(* IEC 61131-3 sources: verifaps-lib/share/xPPU (part 20) *)

(* ---- PLCOpenXML_Scenario_21.st ---- *)
// Extracted from file:/home/weigl/work/verifaps-lib/lang/../share/xPPU/PLCOpenXML_Scenario_21.xml on Wed Feb 05 17:44:48 CET 2020

FUNCTION_BLOCK A_to_V_Transducer

    VAR
        AI_AmperToVolt : INT;
    END_VAR

END_FUNCTION_BLOCK

FUNCTION_BLOCK BistableCylinder

    VAR_OUTPUT
        Extended : BOOL;
        Retracted : BOOL;
    END_VAR

    VAR
        DI_Extended : BOOL;
        DI_Retracted : BOOL;
        DO_Extend : BOOL;
        DO_Retract : BOOL;
        DI_BoundaryPressure : BOOL;
        DI_VacuumBoundaryPressure : BOOL;
        DI_VacuumBoundaryFlowPressure : BOOL;
        AI_PressureSensor : INT;
        AI_FlowPressure : INT;
        AI_PositionTransmitter : INT;
        SFCInit : BOOL;
        SFCReset : BOOL;
    END_VAR
    ACTION ACT_Extend

        INITIAL_STEP Init_ACT_Extend : (*Local Id: 0 *)
        END_STEP

        STEP Extend_Cylinder : (*Local Id: 3 *)
        END_STEP

        STEP SetExtended : (*Local Id: 9 *)
        END_STEP
        TRANSITION FROM (Init_ACT_Extend) TO (Extend_Cylinder) := (NOT Extended AND NOT GVL.IsSFCResetting); END_TRANSITION
        TRANSITION FROM (Extend_Cylinder) TO (SetExtended) := (DI_Extended); END_TRANSITION
        TRANSITION FROM (SetExtended) TO (Init_ACT_Extend) := (Extended); END_TRANSITION
    END_ACTION
    ACTION ACT_Retract

        INITIAL_STEP Init_ACT_Retract : (*Local Id: 0 *)
        END_STEP

        STEP Retract_Cylinder : (*Local Id: 3 *)
        END_STEP

        STEP SetRetacted : (*Local Id: 9 *)
        END_STEP
        TRANSITION FROM (Init_ACT_Retract) TO (Retract_Cylinder) := (NOT Retracted AND NOT GVL.IsSFCResetting); END_TRANSITION
        TRANSITION FROM (Retract_Cylinder) TO (SetRetacted) := (DI_Retracted); END_TRANSITION
        TRANSITION FROM (SetRetacted) TO (Init_ACT_Retract) := (Retracted); END_TRANSITION
    END_ACTION

END_FUNCTION_BLOCK

FUNCTION_BLOCK Crane

    VAR_INPUT
        LiftingCylinder : MonostableCylinder;
        Gripper : VacuumGripper;
        Table : TurningTable;
        SoftwareEmergency : BOOL;
        Check_Stack_WPProvided : BOOL;
        Check_Stack_WPType_Black : BOOL;
        Check_Stack_WPType_White : BOOL;
        Check_Stack_WPType_Metallic : BOOL;
        Check_LargeSortingConveyor_IsSorting : BOOL;
        Check_LargeSortingConveyor_AutomaticExecuteCompleted : BOOL;
        Check_Stamp_IsStamping : BOOL;
        Check_Stamp_WPAvailable : BOOL;
        Check_Stamp_AutomaticExecuteCompleted : BOOL;
        Check_RefillConveyor_IsSending : BOOL;
        Check_EngineStop : BOOL;
        SFCReset : BOOL;
    END_VAR

    VAR_OUTPUT
        InitCompleted : BOOL;
        AutomaticExecuteCompleted : BOOL;
        Conveyor_AllowedToOperate : BOOL;
        Stamp_AllowedToOperate : BOOL;
        WPPickedUp : BOOL;
        EmergencyHandled : BOOL;
    END_VAR

    VAR
        CraneSpeed : INT;
        WPPutDown : BOOL;
        ReachedStack : BOOL;
        ReachedConveyor : BOOL;
        ReachedStamp : BOOL;
        WPType_White : BOOL;
        WPType_Black : BOOL;
        WPType_Metallic : BOOL;
        WPWeight_Light : BOOL;
        WPWeight_Medium : BOOL;
        WPWeight_Heavy : BOOL;
        SFCInit : BOOL;
    END_VAR
    ACTION Reset_ConveyorAllowedToOperate

        Conveyor_AllowedToOperate := FALSE;
    END_ACTION
    ACTION Reset_StampAllowedToOperate

        Stamp_AllowedToOperate := FALSE;
    END_ACTION
    ACTION Reset_Variables

        InitCompleted := FALSE;
        AutomaticExecuteCompleted := FALSE;
        Conveyor_AllowedToOperate := FALSE;
        Stamp_AllowedToOperate := FALSE;

        WPPickedUp := FALSE;
        WPPutDown := FALSE;
        ReachedStack := FALSE;
        ReachedConveyor := FALSE;
        ReachedStamp := FALSE;
        WPType_White := FALSE;
        WPType_Black := FALSE;
        WPType_Metallic := FALSE;
        WPWeight_Light := FALSE;
        WPWeight_Medium := FALSE;
        WPWeight_Heavy := FALSE;
    END_ACTION
    ACTION Set_ConveyorAllowedToOperate

        Conveyor_AllowedToOperate := TRUE;
    END_ACTION
    ACTION Set_StampAllowedToOperate

        Stamp_AllowedToOperate := TRUE;
    END_ACTION
    ACTION Set_WPTypeEqualsStack

        WPType_White:=Main.Stack_WPType_White;
        WPType_Black:=Main.Stack_WPType_Black;
        WPType_Metallic:=Main.Stack_WPType_Metallic;
        WPWeight_Light:=Main.Stack_WPWeight_Light;
        WPWeight_Medium:=Main.Stack_WPWeight_Medium;
        WPWeight_Heavy:=Main.Stack_WPWeight_Heavy;
    END_ACTION
    ACTION Set_WPTypeEqualsStamp

        WPType_White:=Main.Stamp_WPType_White;
        WPType_Black:=Main.Stamp_WPType_Black;
        WPType_Metallic:=Main.Stamp_WPType_Metallic;
        WPWeight_Light:=Main.Stamp_WPWeight_Light;
        WPWeight_Medium:=Main.Stamp_WPWeight_Medium;
        WPWeight_Heavy:=Main.Stamp_WPWeight_Heavy;
    END_ACTION
    ACTION ACT_MoveToConveyor

        INITIAL_STEP Init_MoveToConveyor : (*Local Id: 0 *)
        END_STEP

        STEP DecideHowToMoveCrane : (*Local Id: 3 *)
        END_STEP

        STEP Turn_CounterClockwise_MTC : (*Local Id: 7 *)
            Table.Motor.ACT_TurnCounterclockwise(N);
        END_STEP

        STEP Turn_CLockwise_MTC : (*Local Id: 13 *)
            Table.Motor.ACT_TurnClockwise(N);
        END_STEP

        STEP First_Turn_CounterC : (*Local Id: 18 *)
            Table.Motor.ACT_TurnCounterclockwise(N);
        END_STEP

        STEP Second_Turn_Clockwise : (*Local Id: 24 *)
            Table.Motor.ACT_TurnClockwise(N);
        END_STEP

        STEP StopCrane : (*Local Id: 30 *)
            Table.Motor.ACT_Stop(N);
        END_STEP

        STEP SetReachedConveyor : (*Local Id: 33 *)
        END_STEP
        TRANSITION FROM (DecideHowToMoveCrane) TO (Turn_CounterClockwise_MTC) := (Table.AtStack.DI_SwitchTrue); END_TRANSITION
        TRANSITION FROM (DecideHowToMoveCrane) TO (Turn_CLockwise_MTC) := (Table.AtStamp.DI_SwitchTrue); END_TRANSITION
        TRANSITION FROM (DecideHowToMoveCrane) TO (First_Turn_CounterC) := (NOT (Table.AtStack.DI_SwitchTrue AND Table.AtStamp.DI_SwitchTrue)); END_TRANSITION
        TRANSITION FROM (DecideHowToMoveCrane) TO (Turn_CLockwise_MTC) := (Table.AtStamp.DI_SwitchTrue); END_TRANSITION
        TRANSITION FROM (DecideHowToMoveCrane) TO (First_Turn_CounterC) := (NOT (Table.AtStack.DI_SwitchTrue AND Table.AtStamp.DI_SwitchTrue)); END_TRANSITION
        TRANSITION FROM (First_Turn_CounterC) TO (StopCrane) := (Table.AtConveyor.DI_SwitchTrue); END_TRANSITION
        TRANSITION FROM (First_Turn_CounterC) TO (Second_Turn_Clockwise) := (First_Turn_CounterC.t>T#8s AND Not Table.AtConveyor.DI_SwitchTrue); END_TRANSITION
        TRANSITION FROM (First_Turn_CounterC) TO (StopCrane) := (Table.AtConveyor.DI_SwitchTrue); END_TRANSITION
        TRANSITION FROM (Second_Turn_Clockwise) TO (StopCrane) := (Table.AtConveyor.DI_SwitchTrue); END_TRANSITION
        TRANSITION FROM (Turn_CLockwise_MTC) TO (StopCrane) := (Table.AtConveyor.DI_SwitchTrue); END_TRANSITION
        TRANSITION FROM (First_Turn_CounterC) TO (StopCrane) := (Table.AtConveyor.DI_SwitchTrue); END_TRANSITION
        TRANSITION FROM (Second_Turn_Clockwise) TO (StopCrane) := (Table.AtConveyor.DI_SwitchTrue); END_TRANSITION
        TRANSITION FROM (Turn_CounterClockwise_MTC) TO (StopCrane) := (Table.AtConveyor.DI_SwitchTrue); END_TRANSITION
        TRANSITION FROM (Turn_CLockwise_MTC) TO (StopCrane) := (Table.AtConveyor.DI_SwitchTrue); END_TRANSITION
        TRANSITION FROM (First_Turn_CounterC) TO (StopCrane) := (Table.AtConveyor.DI_SwitchTrue); END_TRANSITION
        TRANSITION FROM (Second_Turn_Clockwise) TO (StopCrane) := (Table.AtConveyor.DI_SwitchTrue); END_TRANSITION
        TRANSITION FROM (Init_MoveToConveyor) TO (DecideHowToMoveCrane) := (NOT GVL.IsSFCResetting); END_TRANSITION
        TRANSITION FROM (StopCrane) TO (SetReachedConveyor) := (Table.Motor.Stopped); END_TRANSITION
        TRANSITION FROM (SetReachedConveyor) TO (Init_MoveToConveyor) := (ReachedConveyor); END_TRANSITION
    END_ACTION
    ACTION ACT_MoveToStack

        INITIAL_STEP Init_MoveToMagazine : (*Local Id: 0 *)
        END_STEP

        STEP Turn_Clockwise_MTM : (*Local Id: 3 *)
            Table.Motor.ACT_TurnClockwise(N);
        END_STEP

        STEP Turn_Counterclockwise : (*Local Id: 9 *)
            Table.Motor.ACT_TurnCounterclockwise(N);
        END_STEP

        STEP StopCrane : (*Local Id: 13 *)
            Table.Motor.ACT_Stop(N);
        END_STEP

        STEP SetReachedStack : (*Local Id: 16 *)
        END_STEP
        TRANSITION FROM (Turn_Clockwise_MTM) TO (StopCrane) := (Table.AtStack.DI_SwitchTrue); END_TRANSITION
        TRANSITION FROM (Turn_Clockwise_MTM) TO (Turn_Counterclockwise) := (Turn_Clockwise_MTM.t>T#8s); END_TRANSITION
        TRANSITION FROM (Turn_Clockwise_MTM) TO (StopCrane) := (Table.AtStack.DI_SwitchTrue); END_TRANSITION
        TRANSITION FROM (Turn_Counterclockwise) TO (StopCrane) := (Table.AtStack.DI_SwitchTrue); END_TRANSITION
        TRANSITION FROM (Init_MoveToMagazine) TO (Turn_Clockwise_MTM) := (NOT GVL.IsSFCResetting); END_TRANSITION
        TRANSITION FROM (StopCrane) TO (SetReachedStack) := (Table.Motor.Stopped); END_TRANSITION
        TRANSITION FROM (SetReachedStack) TO (Init_MoveToMagazine) := (ReachedStack); END_TRANSITION
    END_ACTION
    ACTION ACT_MoveToStamp

        INITIAL_STEP Init_MoveToStamp : (*Local Id: 0 *)
        END_STEP

        STEP Turn_CounterClockwise_MTS : (*Local Id: 3 *)
            Table.Motor.ACT_TurnCounterclockwise(N);
        END_STEP

        STEP Turn_Clockwise : (*Local Id: 9 *)
            Table.Motor.ACT_TurnClockwise(N);
        END_STEP

        STEP StopCrane : (*Local Id: 13 *)
            Table.Motor.ACT_Stop(N);
        END_STEP

        STEP SetReachedStamp : (*Local Id: 16 *)
        END_STEP
        TRANSITION FROM (Turn_CounterClockwise_MTS) TO (StopCrane) := (Table.AtStamp.DI_SwitchTrue); END_TRANSITION
        TRANSITION FROM (Turn_CounterClockwise_MTS) TO (Turn_Clockwise) := (Turn_CounterClockwise_MTS.t>T#8s); END_TRANSITION
        TRANSITION FROM (Turn_CounterClockwise_MTS) TO (StopCrane) := (Table.AtStamp.DI_SwitchTrue); END_TRANSITION
        TRANSITION FROM (Turn_Clockwise) TO (StopCrane) := (Table.AtStamp.DI_SwitchTrue); END_TRANSITION
        TRANSITION FROM (Init_MoveToStamp) TO (Turn_CounterClockwise_MTS) := (NOT GVL.IsSFCResetting); END_TRANSITION
        TRANSITION FROM (StopCrane) TO (SetReachedStamp) := (Table.Motor.Stopped); END_TRANSITION
        TRANSITION FROM (SetReachedStamp) TO (Init_MoveToStamp) := (ReachedStamp); END_TRANSITION
    END_ACTION
    ACTION ACT_PickUpWP

        INITIAL_STEP Init_PickUpWP : (*Local Id: 0 *)
        END_STEP

        STEP Crane_Down : (*Local Id: 3 *)
            LiftingCylinder.ACT_Extend(N);
        END_STEP

        STEP SetWPType : (*Local Id: 6 *)
        END_STEP

        STEP WPType_Is_WPTypeStack : (*Local Id: 10 *)
            Set_WPTypeEqualsStack(N);
        END_STEP

        STEP WPType_Is_WPTypeStamp : (*Local Id: 15 *)
            Set_WPTypeEqualsStamp(N);
        END_STEP

        STEP Turn_On_Vacuum_PWU : (*Local Id: 19 *)
            Gripper.ACT_Intake(N);
        END_STEP

        STEP Crane_Up : (*Local Id: 23 *)
            LiftingCylinder.ACT_Retract(N);
        END_STEP

        STEP Error : (*Local Id: 28 *)
        END_STEP

        STEP SetWPPickedUp : (*Local Id: 35 *)
        END_STEP
        TRANSITION FROM (SetWPType) TO (WPType_Is_WPTypeStack) := (ReachedStack); END_TRANSITION
        TRANSITION FROM (SetWPType) TO (WPType_Is_WPTypeStamp) := (ReachedStamp); END_TRANSITION
        TRANSITION FROM (Turn_On_Vacuum_PWU) TO (Crane_Up) := (Gripper.Intaken); END_TRANSITION
        TRANSITION FROM (Turn_On_Vacuum_PWU) TO (Error) := (Turn_On_Vacuum_PWU.t>T#2s AND NOT Gripper.Intaken); END_TRANSITION
        TRANSITION FROM (WPType_Is_WPTypeStack) TO (Turn_On_Vacuum_PWU) := (WPWeight_Heavy=Main.Stack_WPWeight_Heavy); END_TRANSITION
        TRANSITION FROM (WPType_Is_WPTypeStamp) TO (Turn_On_Vacuum_PWU) := (WPWeight_Heavy=Main.Stamp_WPWeight_Heavy); END_TRANSITION
        TRANSITION FROM (Crane_Up) TO (SetWPPickedUp) := (LiftingCylinder.Retracted); END_TRANSITION
        TRANSITION FROM (Init_PickUpWP) TO (Crane_Down) := (NOT GVL.IsSFCResetting); END_TRANSITION
        TRANSITION FROM (Crane_Down) TO (SetWPType) := (LiftingCylinder.Extended); END_TRANSITION
        TRANSITION FROM (Error) TO (Init_PickUpWP) := (SoftwareEmergency); END_TRANSITION
        TRANSITION FROM (SetWPPickedUp) TO (Init_PickUpWP) := (WPPickedUp); END_TRANSITION
    END_ACTION
    ACTION ACT_PutDownWP

        INITIAL_STEP Init_PutWPDown : (*Local Id: 0 *)
        END_STEP

        STEP WPWeight_Choice : (*Local Id: 3 *)
        END_STEP

        STEP WPLight : (*Local Id: 7 *)
        END_STEP

        STEP WPMedium : (*Local Id: 12 *)
        END_STEP

        STEP WPHeavy : (*Local Id: 17 *)
        END_STEP

        STEP Lower_Crane_PWD : (*Local Id: 21 *)
            LiftingCylinder.ACT_Extend(N);
        END_STEP

        STEP Put_WP_Down_1 : (*Local Id: 24 *)
            Gripper.ACT_Release(N);
        END_STEP

        STEP Crane_Up : (*Local Id: 27 *)
            LiftingCylinder.ACT_Retract(N);
        END_STEP

        STEP SetWPPutDown : (*Local Id: 30 *)
        END_STEP
        TRANSITION FROM (WPWeight_Choice) TO (WPLight) := (WPWeight_Light); END_TRANSITION
        TRANSITION FROM (WPWeight_Choice) TO (WPMedium) := (WPWeight_Medium); END_TRANSITION
        TRANSITION FROM (WPWeight_Choice) TO (WPHeavy) := (WPWeight_Heavy); END_TRANSITION
        TRANSITION FROM (WPLight) TO (Lower_Crane_PWD) := (WPLight.t>T#0ms); END_TRANSITION
        TRANSITION FROM (WPMedium) TO (Lower_Crane_PWD) := (WPMedium.t>T#1000ms); END_TRANSITION
        TRANSITION FROM (WPHeavy) TO (Lower_Crane_PWD) := (WPHeavy.t>T#2000ms); END_TRANSITION
        TRANSITION FROM (Init_PutWPDown) TO (WPWeight_Choice) := (NOT GVL.IsSFCResetting); END_TRANSITION
        TRANSITION FROM (Lower_Crane_PWD) TO (Put_WP_Down_1) := (LiftingCylinder.Extended); END_TRANSITION
        TRANSITION FROM (Put_WP_Down_1) TO (Crane_Up) := (Gripper.Released); END_TRANSITION
        TRANSITION FROM (Crane_Up) TO (SetWPPutDown) := (LiftingCylinder.Retracted); END_TRANSITION
        TRANSITION FROM (SetWPPutDown) TO (Init_PutWPDown) := (WPPutDown); END_TRANSITION
    END_ACTION
    ACTION ACT_AutomaticExecute

        INITIAL_STEP ACT_AutomaticExecute_Init : (*Local Id: 0 *)
        END_STEP

        STEP Waiting_For_Stack_To_Provide_WP : (*Local Id: 3 *)
        END_STEP

        STEP Check_WP_Type : (*Local Id: 6 *)
        END_STEP

        STEP Crane_To_Stamp_1 : (*Local Id: 10 *)
            ACT_MoveToStack(N);
        END_STEP

        STEP Pick_Up_WP_1 : (*Local Id: 13 *)
            ACT_PickUpWP(N);
        END_STEP

        STEP Check_RC_1 : (*Local Id: 16 *)
        END_STEP

        STEP Crane_Turning_To_Conveyor_1 : (*Local Id: 19 *)
            ACT_MoveToConveyor(N);
        END_STEP

        STEP Putting_Down_WP_1 : (*Local Id: 22 *)
            ACT_PutDownWP(N);
        END_STEP

        STEP Short_Delay : (*Local Id: 25 *)
        END_STEP

        STEP Sort_WP : (*Local Id: 28 *)
            Set_ConveyorAllowedToOperate(P0);
            Reset_ConveyorAllowedToOperate(P1);
        END_STEP

        STEP CheckStamp_WPAvailable : (*Local Id: 31 *)
        END_STEP

        STEP WP_Should_Be_Stamped : (*Local Id: 41 *)
        END_STEP

        STEP Crane_Turning_To_Stack_1 : (*Local Id: 45 *)
            ACT_MoveToStack(N);
        END_STEP

        STEP Crane_Pick_Up_Wp_2 : (*Local Id: 48 *)
            ACT_PickUpWP(N);
        END_STEP

        STEP Check_RC_2 : (*Local Id: 51 *)
        END_STEP

        STEP Crane_Turning_To_Stamp_2 : (*Local Id: 54 *)
            ACT_MoveToStamp(N);
        END_STEP

        STEP Crane_Put_Down_WP_2 : (*Local Id: 57 *)
            ACT_PutDownWP(N);
        END_STEP

        STEP Stamping_WP : (*Local Id: 60 *)
            Set_StampAllowedToOperate(P0);
        END_STEP

        STEP CheckStamp_AutomaticExecuteCompleted : (*Local Id: 68 *)
            Reset_StampAllowedToOperate(P1);
        END_STEP

        STEP Crane_Turning_To_Stamp_3 : (*Local Id: 73 *)
            ACT_MoveToStamp(N);
        END_STEP
        TRANSITION FROM (Check_WP_Type) TO (Crane_To_Stamp_1) := (Check_Stack_WPType_Black); END_TRANSITION
        TRANSITION FROM (Check_WP_Type) TO (WP_Should_Be_Stamped) := (Check_Stack_WPType_Metallic OR Check_Stack_WPType_White); END_TRANSITION
        TRANSITION FROM (CheckStamp_WPAvailable) TO (Waiting_For_Stack_To_Provide_WP) := (NOT Check_Stamp_WPAvailable); END_TRANSITION
        TRANSITION FROM (CheckStamp_WPAvailable) TO (Crane_Turning_To_Stamp_3) := (Check_Stamp_WPAvailable); END_TRANSITION
        TRANSITION FROM (WP_Should_Be_Stamped) TO (Crane_Turning_To_Stack_1) := (NOT Check_Stamp_IsStamping); END_TRANSITION
        TRANSITION FROM (WP_Should_Be_Stamped) TO (Crane_Turning_To_Stamp_3) := (Check_Stamp_IsStamping); END_TRANSITION
        TRANSITION FROM (Stamping_WP) TO (CheckStamp_AutomaticExecuteCompleted) := (Check_Stack_WPType_Metallic OR Check_Stack_WPType_White); END_TRANSITION
        TRANSITION FROM (Stamping_WP) TO (Crane_To_Stamp_1) := (Check_Stack_WPType_Black); END_TRANSITION
        TRANSITION FROM (CheckStamp_WPAvailable) TO (Waiting_For_Stack_To_Provide_WP) := (NOT Check_Stamp_WPAvailable); END_TRANSITION
        TRANSITION FROM (Stamping_WP) TO (CheckStamp_AutomaticExecuteCompleted) := (Check_Stack_WPType_Metallic OR Check_Stack_WPType_White); END_TRANSITION
        TRANSITION FROM (CheckStamp_AutomaticExecuteCompleted) TO (Pick_Up_WP_1) := (Check_Stamp_AutomaticExecuteCompleted); END_TRANSITION
        TRANSITION FROM (Crane_Turning_To_Stamp_3) TO (Pick_Up_WP_1) := (ReachedStamp AND NOT Check_Stamp_AutomaticExecuteCompleted); END_TRANSITION
        TRANSITION FROM (CheckStamp_WPAvailable) TO (Waiting_For_Stack_To_Provide_WP) := (NOT Check_Stamp_WPAvailable); END_TRANSITION
        TRANSITION FROM (ACT_AutomaticExecute_Init) TO (Waiting_For_Stack_To_Provide_WP) := (NOT AutomaticExecuteCompleted AND NOT GVL.IsSFCResetting); END_TRANSITION
        TRANSITION FROM (Waiting_For_Stack_To_Provide_WP) TO (Check_WP_Type) := (Check_Stack_WPProvided); END_TRANSITION
        TRANSITION FROM (Crane_To_Stamp_1) TO (Pick_Up_WP_1) := (ReachedStack); END_TRANSITION
        TRANSITION FROM (Pick_Up_WP_1) TO (Check_RC_1) := (WPPickedUp); END_TRANSITION
        TRANSITION FROM (Check_RC_1) TO (Crane_Turning_To_Conveyor_1) := (NOT Check_RefillConveyor_IsSending AND Check_Rc_1.t>T#250ms); END_TRANSITION
        TRANSITION FROM (Crane_Turning_To_Conveyor_1) TO (Putting_Down_WP_1) := (ReachedConveyor AND NOT Check_LargeSortingConveyor_IsSorting); END_TRANSITION
        TRANSITION FROM (Putting_Down_WP_1) TO (Short_Delay) := (WPPutDown); END_TRANSITION
        TRANSITION FROM (Short_Delay) TO (Sort_WP) := (Short_Delay.t>T#50ms); END_TRANSITION
        TRANSITION FROM (Sort_WP) TO (CheckStamp_WPAvailable) := (Check_LargeSortingConveyor_AutomaticExecuteCompleted); END_TRANSITION
        TRANSITION FROM (Crane_Turning_To_Stack_1) TO (Crane_Pick_Up_Wp_2) := (ReachedStack); END_TRANSITION
        TRANSITION FROM (Crane_Pick_Up_Wp_2) TO (Check_RC_2) := (WPPickedUp); END_TRANSITION
        TRANSITION FROM (Check_RC_2) TO (Crane_Turning_To_Stamp_2) := (NOT Check_RefillConveyor_IsSending AND Check_Rc_2.t>T#250ms); END_TRANSITION
        TRANSITION FROM (Crane_Turning_To_Stamp_2) TO (Crane_Put_Down_WP_2) := (ReachedStamp); END_TRANSITION
        TRANSITION FROM (Crane_Put_Down_WP_2) TO (Stamping_WP) := (WPPutDown); END_TRANSITION
    END_ACTION
    ACTION ACT_EmergencyStop

        INITIAL_STEP Crane_ACT_EmergencyStop_Init : (*Local Id: 0 *)
        END_STEP

        STEP ResetVariables : (*Local Id: 3 *)
            Reset_Variables(N);
        END_STEP

        STEP StopCrane : (*Local Id: 6 *)
            Table.Motor.ACT_Stop(N);
        END_STEP

        STEP Turn_Vacuum_Off : (*Local Id: 12 *)
            Gripper.ACT_Release(N);
        END_STEP

        STEP Retract_LiftingCylinder : (*Local Id: 16 *)
            LiftingCylinder.ACT_Retract(N);
        END_STEP

        STEP Crane_EmergencyHandled : (*Local Id: 19 *)
        END_STEP
        TRANSITION FROM (StopCrane) TO (Retract_LiftingCylinder) := (Table.Motor.Stopped AND Gripper.Intaken); END_TRANSITION
        TRANSITION FROM (StopCrane) TO (Turn_Vacuum_Off) := (Table.Motor.Stopped AND NOT Gripper.Intaken); END_TRANSITION
        TRANSITION FROM (StopCrane) TO (Retract_LiftingCylinder) := (Table.Motor.Stopped AND Gripper.Intaken); END_TRANSITION
        TRANSITION FROM (Turn_Vacuum_Off) TO (Retract_LiftingCylinder) := (Gripper.Released); END_TRANSITION
        TRANSITION FROM (Crane_ACT_EmergencyStop_Init) TO (ResetVariables) := (NOT EmergencyHandled AND NOT GVL.IsSFCResetting); END_TRANSITION
        TRANSITION FROM (ResetVariables) TO (StopCrane) := (NOT InitCompleted AND NOT AutomaticExecuteCompleted); END_TRANSITION
        TRANSITION FROM (Retract_LiftingCylinder) TO (Crane_EmergencyHandled) := (LiftingCylinder.Retracted); END_TRANSITION
        TRANSITION FROM (Crane_EmergencyHandled) TO (Crane_ACT_EmergencyStop_Init) := (EmergencyHandled); END_TRANSITION
    END_ACTION
    ACTION ACT_Init

        INITIAL_STEP Crane_ACT_Init : (*Local Id: 0 *)
        END_STEP

        STEP Crane_MoveUp_Init : (*Local Id: 3 *)
            LiftingCylinder.ACT_Retract(N);
        END_STEP

        STEP WPAllreadyPickedUp : (*Local Id: 9 *)
        END_STEP

        STEP Turn_To_Conveyor : (*Local Id: 14 *)
            ACT_MoveToConveyor(N);
        END_STEP

        STEP Put_WP_On_Conveyor_Init : (*Local Id: 17 *)
            ACT_PutDownWP(N);
        END_STEP

        STEP Is_WP_At_Stamp : (*Local Id: 23 *)
        END_STEP

        STEP Turn_To_Stamp_Init : (*Local Id: 29 *)
            ACT_MoveToStamp(N);
        END_STEP

        STEP PicWPFromStampUp : (*Local Id: 32 *)
            ACT_PickUpWP(N);
        END_STEP

        STEP SetInitCompleted : (*Local Id: 37 *)
        END_STEP
        TRANSITION FROM (Crane_MoveUp_Init) TO (Is_WP_At_Stamp) := (LiftingCylinder.Retracted AND NOT Gripper.VacuumSwitch.DI_TakenIn); END_TRANSITION
        TRANSITION FROM (Crane_MoveUp_Init) TO (WPAllreadyPickedUp) := (LiftingCylinder.Retracted AND Gripper.VacuumSwitch.DI_TakenIn); END_TRANSITION
        TRANSITION FROM (Is_WP_At_Stamp) TO (SetInitCompleted) := (NOT Check_Stamp_WPAvailable); END_TRANSITION
        TRANSITION FROM (Is_WP_At_Stamp) TO (Turn_To_Stamp_Init) := (Check_Stamp_WPAvailable); END_TRANSITION
        TRANSITION FROM (Crane_MoveUp_Init) TO (Is_WP_At_Stamp) := (LiftingCylinder.Retracted AND NOT Gripper.VacuumSwitch.DI_TakenIn); END_TRANSITION
        TRANSITION FROM (Put_WP_On_Conveyor_Init) TO (Is_WP_At_Stamp) := (WPPutDown); END_TRANSITION
        TRANSITION FROM (Is_WP_At_Stamp) TO (SetInitCompleted) := (NOT Check_Stamp_WPAvailable); END_TRANSITION
        TRANSITION FROM (Crane_ACT_Init) TO (Crane_MoveUp_Init) := (NOT InitCompleted AND NOT GVL.IsSFCResetting); END_TRANSITION
        TRANSITION FROM (WPAllreadyPickedUp) TO (Turn_To_Conveyor) := (WPPickedUp); END_TRANSITION
        TRANSITION FROM (Turn_To_Conveyor) TO (Put_WP_On_Conveyor_Init) := (ReachedConveyor); END_TRANSITION
        TRANSITION FROM (Turn_To_Stamp_Init) TO (PicWPFromStampUp) := (ReachedStamp); END_TRANSITION
        TRANSITION FROM (PicWPFromStampUp) TO (Turn_To_Conveyor) := (WPPickedUp); END_TRANSITION
        TRANSITION FROM (SetInitCompleted) TO (Crane_ACT_Init) := (InitCompleted); END_TRANSITION
    END_ACTION

    Check_Stack_WPProvided := Main.Stack_WPProvided;
    Check_Stack_WPType_Black := Main.Stack_WPType_Black;
    Check_Stack_WPType_White := Main.Stack_WPType_White;
    Check_Stack_WPType_Metallic := Main.Stack_WPType_Metallic;
    Check_LargeSortingConveyor_IsSorting := Main.LargeSortingConveyor_IsSorting;
    Check_LargeSortingConveyor_AutomaticExecuteCompleted := Main.LargeSortingConveyor_AutomaticExecuteCompleted;
    Check_Stamp_IsStamping := Main.Stamp_IsStamping;
    Check_Stamp_WPAvailable := Main.Stamp_WPAvailable;
    Check_Stamp_AutomaticExecuteCompleted := Main.Stamp_AutomaticExecuteCompleted;
    Check_RefillConveyor_IsSending := Main.Check_RefillConveyor_IsSending;
    Check_EngineStop := MAIN.PPU_EngineStop;
    IF Check_EngineStop THEN
    	Table.Motor.ACT_Stop();
    END_IF
END_FUNCTION_BLOCK

FUNCTION_BLOCK EnergyMonitor

    VAR
        BK_1_6_Wattmeter : Wattmeter;
        BK_2_3_7_Wattmeter : Wattmeter;
        BK_4_5_8_9_10_11_Wattmeter : Wattmeter;
        GearPoint_80l_min : GearPointFlowSensor;
        GearPoint_120l_min : GearPointFlowSensor;
        PressureSensor_4bar : PressureSensor_4bar;
        Flow_2to200l_min : FlowSensor;
        Transducer_0to10AC_0to10V : A_to_V_Transducer;
        ExtSensor_0to10V : V_Sensor;
        PressureSensor : PressureSensor;
        SmallContacter_left : ProtectiveContact;
        SmallContacter_right : ProtectiveContact;
        ChangeoverMagnetVaveRelay : MagnetValve;
    END_VAR

END_FUNCTION_BLOCK

FUNCTION_BLOCK FlowSensor

    VAR
        AI_Flow : INT;
    END_VAR

END_FUNCTION_BLOCK

FUNCTION_BLOCK GearPointFlowSensor

    VAR
        DI_ReachedGearPoint : BOOL;
    END_VAR

END_FUNCTION_BLOCK

FUNCTION_BLOCK InductiveSensor

    VAR
        DI_WPMetallic : BOOL;
    END_VAR

END_FUNCTION_BLOCK

FUNCTION_BLOCK InductiveSwitch

    VAR
        DI_InductiveSwitchTrue : BOOL;
    END_VAR

END_FUNCTION_BLOCK

FUNCTION_BLOCK LargeSortingConveyor

    VAR_INPUT
        Panel : OperationPanel;
        Motor : Motor;
        Seperator1 : MonostableCylinder;
        Seperator2 : MonostableCylinder;
        PsBeginning : PresenceSensor;
        OptRamp1 : OpticalSensor;
        IndRamp1 : InductiveSensor;
        Ramp1 : Ramp;
        UltrasonicSensor : UltrasonicSensor;
        Switch : Switch;
        OptRamp2 : OpticalSensor;
        IndRamp2 : InductiveSensor;
        Ramp2 : Ramp;
        OptEnd : OpticalSensor;
        Ramp3 : Ramp;
        OptBeginning : OpticalSensor;
        Check_AllowedToOperate : BOOL;
        Check_FollowConveyorInitCompleted : BOOL;
        Check_FollowConveyorAutoamticExecuteCompleted : BOOL;
        Check_EngineStop : BOOL;
        SFCReset : BOOL;
    END_VAR

    VAR_OUTPUT
        StartButton : BOOL;
        ManuelMode : BOOL;
        AutomaticMode : BOOL;
        InitCompleted : BOOL;
        FollowConveyor_AllowedToInit : BOOL;
        FollowConveyor_AllowedToOperate : BOOL;
        NumberOfWPsAtConveyor : USINT;
        AutomaticExecuteCompleted : BOOL;
        EmergencyStop : BOOL;
        EmergencyHandled : BOOL;
        IsSorting : BOOL;
    END_VAR

    VAR
        ConveyorSpeed : INT;
        WPSorted : BOOL;
        WPTypeChecked : BOOL;
        TargetChanged : BOOL;
        WPType_White : BOOL;
        WPType_Black : BOOL;
        WPType_Metallic : BOOL;
        CurrentTarget_Ramp1 : BOOL;
        CurrentTarget_Conveyor : BOOL;
        CurrentTarget_Ramp2 : BOOL;
        CurrentTarget_Ramp3 : BOOL;
        Priority_White : UINT;
        Priority_Black : UINT;
        Priority_Metallic : UINT;
        SFCInit : BOOL;
    END_VAR
    ACTION Reset_FollowConveyorAllowedToOperate

        FollowConveyor_AllowedToOperate := FALSE;
    END_ACTION
    ACTION Reset_Variables

        InitCompleted := FALSE;
        FollowConveyor_AllowedToInit := FALSE;
        FollowConveyor_AllowedToOperate := FALSE;
        AutomaticExecuteCompleted := FALSE;
        IsSorting:=FALSE;

        WPSorted:=FALSE;
        WPTypeChecked:=FALSE;
        TargetChanged:=FALSE;
        WPType_White:=FALSE;
        WPType_Black:=FALSE;
        WPType_Metallic:=FALSE;
        CurrentTarget_Ramp1:=FALSE;
        CurrentTarget_Conveyor:=FALSE;
        CurrentTarget_Ramp2:=FALSE;
        CurrentTarget_Ramp3:=FALSE;
    END_ACTION
    ACTION Set_FollowConveyorAllowedToOperate

        FollowConveyor_AllowedToOperate := TRUE;
    END_ACTION
    ACTION Set_OneWP

        NumberOfWPsAtConveyor:=1;
    END_ACTION
    ACTION Set_PriorityBlack

        Priority_Black := 4;
    END_ACTION
    ACTION Set_PriorityMetallic

        Priority_Metallic := 3;
    END_ACTION
    ACTION Set_PriorityWhite

        Priority_White := 1;
    END_ACTION
    ACTION Set_ThreeWP

        NumberOfWPsAtConveyor:=3;
    END_ACTION
    ACTION Set_TwoWP

        NumberOfWPsAtConveyor:=2;
    END_ACTION
    ACTION Set_ZeroWP

        NumberOfWPsAtConveyor:=0;
    END_ACTION
    ACTION ACT_ChangeTarget

        INITIAL_STEP ACT_ChangeTarget_Init : (*Local Id: 0 *)
        END_STEP

        STEP ResetTargets : (*Local Id: 3 *)
        END_STEP

        STEP White : (*Local Id: 13 *)
            Set_PriorityWhite(N);
        END_STEP

        STEP Ramp_1 : (*Local Id: 17 *)
        END_STEP

        STEP Choice_Ramp1Full : (*Local Id: 35 *)
        END_STEP

        STEP Conveyor : (*Local Id: 41 *)
        END_STEP

        STEP Black : (*Local Id: 52 *)
            Set_PriorityBlack(N);
        END_STEP

        STEP Ramp_2 : (*Local Id: 56 *)
        END_STEP

        STEP Choice_Ramp2Full : (*Local Id: 74 *)
        END_STEP

        STEP Metallic : (*Local Id: 86 *)
            Set_PriorityMetallic(N);
        END_STEP

        STEP Ramp_3 : (*Local Id: 90 *)
        END_STEP

        STEP Choice_Ramp3Full : (*Local Id: 105 *)
        END_STEP

        STEP SetTargetChanged : (*Local Id: 115 *)
        END_STEP
        TRANSITION FROM (ResetTargets) TO (White) := (WPType_White); END_TRANSITION
        TRANSITION FROM (ResetTargets) TO (Black) := (WPType_Black); END_TRANSITION
        TRANSITION FROM (ResetTargets) TO (Metallic) := (WPType_Metallic); END_TRANSITION
        TRANSITION FROM (ResetTargets) TO (White) := (WPType_White); END_TRANSITION
        TRANSITION FROM (ResetTargets) TO (Black) := (WPType_Black); END_TRANSITION
        TRANSITION FROM (White) TO (Ramp_1) := (Priority_White=1); END_TRANSITION
        TRANSITION FROM (White) TO (Ramp_2) := (Priority_White=2); END_TRANSITION
        TRANSITION FROM (White) TO (Ramp_3) := (Priority_White=3); END_TRANSITION
        TRANSITION FROM (White) TO (Conveyor) := (Priority_White=4); END_TRANSITION
        TRANSITION FROM (Choice_Ramp1Full) TO (SetTargetChanged) := (NOT Ramp1.RampFull.DI_WPDetected); END_TRANSITION
        TRANSITION FROM (Choice_Ramp1Full) TO (Conveyor) := (Ramp1.RampFull.DI_WPDetected); END_TRANSITION
        TRANSITION FROM (Black) TO (Ramp_2) := (Priority_Black=2); END_TRANSITION
        TRANSITION FROM (Black) TO (Ramp_1) := (Priority_Black=1); END_TRANSITION
        TRANSITION FROM (Black) TO (Ramp_3) := (Priority_Black=3); END_TRANSITION
        TRANSITION FROM (Black) TO (Conveyor) := (Priority_Black=4); END_TRANSITION
        TRANSITION FROM (Choice_Ramp2Full) TO (SetTargetChanged) := (NOT Ramp2.RampFull.DI_WPDetected); END_TRANSITION
        TRANSITION FROM (Choice_Ramp2Full) TO (Conveyor) := (Ramp2.RampFull.DI_WPDetected); END_TRANSITION
        TRANSITION FROM (Metallic) TO (Ramp_3) := (Priority_Metallic=3); END_TRANSITION
        TRANSITION FROM (Metallic) TO (Ramp_2) := (Priority_Metallic=1); END_TRANSITION
        TRANSITION FROM (Metallic) TO (Ramp_3) := (Priority_Metallic=2); END_TRANSITION
        TRANSITION FROM (Choice_Ramp3Full) TO (SetTargetChanged) := (NOT Ramp3.RampFull.DI_WPDetected); END_TRANSITION
        TRANSITION FROM (Choice_Ramp3Full) TO (Ramp_2) := (Ramp3.RampFull.DI_WPDetected); END_TRANSITION
        TRANSITION FROM (Ramp_1) TO (Choice_Ramp1Full) := (CurrentTarget_Ramp1); END_TRANSITION
        TRANSITION FROM (Ramp_2) TO (Choice_Ramp1Full) := (CurrentTarget_Ramp1); END_TRANSITION
        TRANSITION FROM (Ramp_3) TO (Choice_Ramp1Full) := (CurrentTarget_Ramp1); END_TRANSITION
        TRANSITION FROM (Conveyor) TO (Choice_Ramp1Full) := (CurrentTarget_Ramp1); END_TRANSITION
        TRANSITION FROM (Choice_Ramp1Full) TO (SetTargetChanged) := (NOT Ramp1.RampFull.DI_WPDetected); END_TRANSITION
        TRANSITION FROM (Conveyor) TO (SetTargetChanged) := (CurrentTarget_Conveyor); END_TRANSITION
        TRANSITION FROM (Ramp_2) TO (Choice_Ramp2Full) := (CurrentTarget_Ramp2); END_TRANSITION
        TRANSITION FROM (Ramp_1) TO (Choice_Ramp2Full) := (CurrentTarget_Ramp2); END_TRANSITION
        TRANSITION FROM (Ramp_3) TO (Choice_Ramp2Full) := (CurrentTarget_Ramp2); END_TRANSITION
        TRANSITION FROM (Conveyor) TO (Choice_Ramp2Full) := (CurrentTarget_Ramp2); END_TRANSITION
        TRANSITION FROM (Choice_Ramp2Full) TO (SetTargetChanged) := (NOT Ramp2.RampFull.DI_WPDetected); END_TRANSITION
        TRANSITION FROM (Choice_Ramp1Full) TO (SetTargetChanged) := (NOT Ramp1.RampFull.DI_WPDetected); END_TRANSITION
        TRANSITION FROM (Conveyor) TO (SetTargetChanged) := (CurrentTarget_Conveyor); END_TRANSITION
        TRANSITION FROM (Ramp_3) TO (Choice_Ramp3Full) := (CurrentTarget_Ramp3); END_TRANSITION
        TRANSITION FROM (Ramp_2) TO (Choice_Ramp3Full) := (CurrentTarget_Ramp3); END_TRANSITION
        TRANSITION FROM (Ramp_3) TO (Choice_Ramp3Full) := (CurrentTarget_Ramp3); END_TRANSITION
        TRANSITION FROM (Choice_Ramp3Full) TO (SetTargetChanged) := (NOT Ramp3.RampFull.DI_WPDetected); END_TRANSITION
        TRANSITION FROM (Choice_Ramp1Full) TO (SetTargetChanged) := (NOT Ramp1.RampFull.DI_WPDetected); END_TRANSITION
        TRANSITION FROM (Conveyor) TO (SetTargetChanged) := (CurrentTarget_Conveyor); END_TRANSITION
        TRANSITION FROM (ACT_ChangeTarget_Init) TO (ResetTargets) := (NOT TargetChanged AND NOT GVL.IsSFCResetting); END_TRANSITION
        TRANSITION FROM (SetTargetChanged) TO (ACT_ChangeTarget_Init) := (TargetChanged); END_TRANSITION
    END_ACTION
    ACTION ACT_CheckWPType

        INITIAL_STEP Conveyor_ACT_CheckWPType_Init : (*Local Id: 0 *)
        END_STEP

        STEP Reset_WPType : (*Local Id: 3 *)
        END_STEP

        STEP WP_Is_White : (*Local Id: 11 *)
        END_STEP

        STEP WP_Is_Black : (*Local Id: 18 *)
        END_STEP

        STEP WP_Is_Metallic : (*Local Id: 25 *)
        END_STEP

        STEP WP_Type_Checked : (*Local Id: 31 *)
        END_STEP
        TRANSITION FROM (Reset_WPType) TO (WP_Is_White) := (OptRamp1.DI_WPLight AND NOT IndRamp1.DI_WPMetallic); END_TRANSITION
        TRANSITION FROM (Reset_WPType) TO (WP_Is_Black) := (NOT IndRamp1.DI_WPMetallic AND NOT OptRamp1.DI_WPLight); END_TRANSITION
        TRANSITION FROM (Reset_WPType) TO (WP_Is_Metallic) := (IndRamp1.DI_WPMetallic); END_TRANSITION
        TRANSITION FROM (WP_Is_White) TO (WP_Type_Checked) := (WPType_White); END_TRANSITION
        TRANSITION FROM (WP_Is_Black) TO (WP_Type_Checked) := (WPType_Black); END_TRANSITION
        TRANSITION FROM (WP_Is_Metallic) TO (WP_Type_Checked) := (WPType_Metallic); END_TRANSITION
        TRANSITION FROM (Conveyor_ACT_CheckWPType_Init) TO (Reset_WPType) := (NOT WPTypeChecked AND NOT GVL.IsSFCResetting); END_TRANSITION
        TRANSITION FROM (WP_Type_Checked) TO (Conveyor_ACT_CheckWPType_Init) := (WPTypeChecked); END_TRANSITION
    END_ACTION
    ACTION ACT_CountWPsAtConveyor

        INITIAL_STEP Init_ACT_CountWPsAtConveyor : (*Local Id: 0 *)
        END_STEP

        STEP Wait500ms_0 : (*Local Id: 4 *)
        END_STEP

        STEP Zero_WP : (*Local Id: 8 *)
            Set_ZeroWP(N);
        END_STEP

        STEP Wait500ms_1 : (*Local Id: 17 *)
        END_STEP

        STEP One_WP : (*Local Id: 21 *)
            Set_OneWP(N);
        END_STEP

        STEP Wait500ms_2 : (*Local Id: 30 *)
        END_STEP

        STEP Two_WP : (*Local Id: 34 *)
            Set_TwoWP(N);
        END_STEP

        STEP Wait500ms_3 : (*Local Id: 43 *)
        END_STEP

        STEP Three_WP : (*Local Id: 47 *)
            Set_ThreeWP(N);
        END_STEP
        TRANSITION FROM (Init_ACT_CountWPsAtConveyor) TO (Wait500ms_0) := (UltrasonicSensor.AI_UltraSonic>=15200); END_TRANSITION
        TRANSITION FROM (Init_ACT_CountWPsAtConveyor) TO (Wait500ms_1) := (15200>UltrasonicSensor.AI_UltraSonic AND UltrasonicSensor.AI_UltraSonic>=13200); END_TRANSITION
        TRANSITION FROM (Init_ACT_CountWPsAtConveyor) TO (Wait500ms_2) := (13200>UltrasonicSensor.AI_UltraSonic AND UltrasonicSensor.AI_UltraSonic>=8500); END_TRANSITION
        TRANSITION FROM (Init_ACT_CountWPsAtConveyor) TO (Wait500ms_3) := (8500>UltrasonicSensor.AI_UltraSonic AND UltrasonicSensor.AI_UltraSonic>=4000); END_TRANSITION
        TRANSITION FROM (Wait500ms_0) TO (Zero_WP) := (Wait500ms_0.t>T#500ms AND UltrasonicSensor.AI_UltraSonic>=15200); END_TRANSITION
        TRANSITION FROM (Wait500ms_0) TO (Init_ACT_CountWPsAtConveyor) := (Wait500ms_0.t>T#500ms AND NOT UltrasonicSensor.AI_UltraSonic>=15200); END_TRANSITION
        TRANSITION FROM (Wait500ms_1) TO (One_WP) := (Wait500ms_1.t>T#500ms AND (15200>UltrasonicSensor.AI_UltraSonic AND UltrasonicSensor.AI_UltraSonic>=13200)); END_TRANSITION
        TRANSITION FROM (Wait500ms_1) TO (Init_ACT_CountWPsAtConveyor) := (Wait500ms_1.t>T#500ms AND NOT (15200>UltrasonicSensor.AI_UltraSonic AND UltrasonicSensor.AI_UltraSonic>=13200)); END_TRANSITION
        TRANSITION FROM (Wait500ms_2) TO (Two_WP) := (Wait500ms_2.t>T#500ms AND (13200>UltrasonicSensor.AI_UltraSonic AND UltrasonicSensor.AI_UltraSonic>=8500)); END_TRANSITION
        TRANSITION FROM (Wait500ms_2) TO (Init_ACT_CountWPsAtConveyor) := (Wait500ms_2.t>T#500ms AND NOT(13200>UltrasonicSensor.AI_UltraSonic AND UltrasonicSensor.AI_UltraSonic>=8500)); END_TRANSITION
        TRANSITION FROM (Wait500ms_3) TO (Three_WP) := (Wait500ms_3.t>T#500ms AND (8500>UltrasonicSensor.AI_UltraSonic AND UltrasonicSensor.AI_UltraSonic>=4000)); END_TRANSITION
        TRANSITION FROM (Wait500ms_3) TO (Init_ACT_CountWPsAtConveyor) := (Wait500ms_3.t>T#500ms AND NOT(8500>UltrasonicSensor.AI_UltraSonic AND UltrasonicSensor.AI_UltraSonic>=4000)); END_TRANSITION
        TRANSITION FROM (Zero_WP) TO (Init_ACT_CountWPsAtConveyor) := (NumberOfWPsAtConveyor=0); END_TRANSITION
        TRANSITION FROM (One_WP) TO (Init_ACT_CountWPsAtConveyor) := (NumberOfWPsAtConveyor=1); END_TRANSITION
        TRANSITION FROM (Two_WP) TO (Init_ACT_CountWPsAtConveyor) := (NumberOfWPsAtConveyor=2); END_TRANSITION
        TRANSITION FROM (Init_ACT_CountWPsAtConveyor) TO (Init_ACT_CountWPsAtConveyor) := (NumberOfWPsAtConveyor=2); END_TRANSITION
        TRANSITION FROM (Three_WP) TO (Init_ACT_CountWPsAtConveyor) := (NumberOfWPsAtConveyor=3); END_TRANSITION
        TRANSITION FROM (Zero_WP) TO (Init_ACT_CountWPsAtConveyor) := (NumberOfWPsAtConveyor=0); END_TRANSITION
        TRANSITION FROM (One_WP) TO (Init_ACT_CountWPsAtConveyor) := (NumberOfWPsAtConveyor=1); END_TRANSITION
        TRANSITION FROM (Two_WP) TO (Init_ACT_CountWPsAtConveyor) := (NumberOfWPsAtConveyor=2); END_TRANSITION
        TRANSITION FROM (Init_ACT_CountWPsAtConveyor) TO (Init_ACT_CountWPsAtConveyor) := (NumberOfWPsAtConveyor=2); END_TRANSITION
        TRANSITION FROM (Three_WP) TO (Init_ACT_CountWPsAtConveyor) := (NumberOfWPsAtConveyor=3); END_TRANSITION
    END_ACTION
    ACTION ACT_SortWP

        INITIAL_STEP Init_ACT_SortWP : (*Local Id: 0 *)
        END_STEP

        STEP TurnConveyorOn : (*Local Id: 3 *)
        END_STEP

        STEP Wait_Till_Detection : (*Local Id: 9 *)
        END_STEP

        STEP Stop_Conveyor : (*Local Id: 12 *)
            Motor.ACT_Stop(N);
        END_STEP

        STEP Checking_WP_Type : (*Local Id: 15 *)
            ACT_CheckWPType(N);
        END_STEP

        STEP Changing_Target : (*Local Id: 18 *)
            ACT_ChangeTarget(N);
        END_STEP

        STEP TrunConveyorOnAgain : (*Local Id: 21 *)
            Motor.ACT_TurnClockwise(N);
        END_STEP

        STEP TurnConveyorOff_1 : (*Local Id: 25 *)
        END_STEP

        STEP Pusher1_Extending : (*Local Id: 30 *)
            Seperator1.ACT_Extend(N);
        END_STEP

        STEP Pusher1_Retracting : (*Local Id: 33 *)
            Seperator1.ACT_Retract(N);
        END_STEP

        STEP ExtendSwitch : (*Local Id: 38 *)
            Switch.ACT_Extend(N);
        END_STEP

        STEP Transporting_To_Conveyor : (*Local Id: 41 *)
        END_STEP

        STEP AllowFollowConveyorToReceiveWP : (*Local Id: 44 *)
            Set_FollowConveyorAllowedToOperate(P0);
            Reset_FollowConveyorAllowedToOperate(P1);
        END_STEP

        STEP TurnConveyorOff_4 : (*Local Id: 47 *)
            Motor.ACT_Stop(N);
        END_STEP

        STEP RetractSwitch : (*Local Id: 50 *)
            Switch.ACT_Retract(N);
        END_STEP

        STEP TurnConveyorOff_2 : (*Local Id: 55 *)
        END_STEP

        STEP Pusher2_Extending : (*Local Id: 60 *)
            Seperator2.ACT_Extend(N);
        END_STEP

        STEP Pusher2_Retract : (*Local Id: 63 *)
            Seperator2.ACT_Retract(N);
        END_STEP

        STEP TurnConveyorOff_3 : (*Local Id: 68 *)
        END_STEP

        STEP WP_Is_Sorted : (*Local Id: 74 *)
        END_STEP
        TRANSITION FROM (TrunConveyorOnAgain) TO (TurnConveyorOff_1) := (CurrentTarget_Ramp1); END_TRANSITION
        TRANSITION FROM (TrunConveyorOnAgain) TO (ExtendSwitch) := (CurrentTarget_Conveyor); END_TRANSITION
        TRANSITION FROM (TrunConveyorOnAgain) TO (TurnConveyorOff_2) := (CurrentTarget_Ramp2); END_TRANSITION
        TRANSITION FROM (TrunConveyorOnAgain) TO (TurnConveyorOff_3) := (CurrentTarget_Ramp3); END_TRANSITION
        TRANSITION FROM (Pusher1_Retracting) TO (WP_Is_Sorted) := (Seperator1.Retracted); END_TRANSITION
        TRANSITION FROM (RetractSwitch) TO (WP_Is_Sorted) := (Switch.Retracted); END_TRANSITION
        TRANSITION FROM (Pusher2_Retract) TO (WP_Is_Sorted) := (Seperator2.Retracted); END_TRANSITION
        TRANSITION FROM (TurnConveyorOff_3) TO (WP_Is_Sorted) := (Motor.Stopped); END_TRANSITION
        TRANSITION FROM (Init_ACT_SortWP) TO (TurnConveyorOn) := (NOT WPSorted AND NOT GVL.IsSFCResetting); END_TRANSITION
        TRANSITION FROM (TurnConveyorOn) TO (Wait_Till_Detection) := (PsBeginning.DI_WPDetected); END_TRANSITION
        TRANSITION FROM (Wait_Till_Detection) TO (Stop_Conveyor) := (Wait_Till_Detection.t>T#300ms); END_TRANSITION
        TRANSITION FROM (Stop_Conveyor) TO (Checking_WP_Type) := (Motor.Stopped); END_TRANSITION
        TRANSITION FROM (Checking_WP_Type) TO (Changing_Target) := (WPTypeChecked); END_TRANSITION
        TRANSITION FROM (Changing_Target) TO (TrunConveyorOnAgain) := (TargetChanged); END_TRANSITION
        TRANSITION FROM (TurnConveyorOff_1) TO (Pusher1_Extending) := (Motor.Stopped); END_TRANSITION
        TRANSITION FROM (Pusher1_Extending) TO (Pusher1_Retracting) := (Seperator1.Extended); END_TRANSITION
        TRANSITION FROM (ExtendSwitch) TO (Transporting_To_Conveyor) := (Switch.Extended); END_TRANSITION
        TRANSITION FROM (Transporting_To_Conveyor) TO (AllowFollowConveyorToReceiveWP) := (Transporting_To_Conveyor.t>T#1500ms); END_TRANSITION
        TRANSITION FROM (AllowFollowConveyorToReceiveWP) TO (TurnConveyorOff_4) := (Check_FollowConveyorAutoamticExecuteCompleted); END_TRANSITION
        TRANSITION FROM (TurnConveyorOff_4) TO (RetractSwitch) := (Motor.Stopped); END_TRANSITION
        TRANSITION FROM (TurnConveyorOff_2) TO (Pusher2_Extending) := (Motor.Stopped); END_TRANSITION
        TRANSITION FROM (Pusher2_Extending) TO (Pusher2_Retract) := (Seperator2.Extended); END_TRANSITION
        TRANSITION FROM (WP_Is_Sorted) TO (Init_ACT_SortWP) := (WPSorted); END_TRANSITION
    END_ACTION
    ACTION ACT_AutomaticExecute

        INITIAL_STEP LargeSortingConveyor_ACT_AutomaticExecute_Init : (*Local Id: 0 *)
        END_STEP

        STEP Interstep : (*Local Id: 3 *)
        END_STEP

        STEP Sort_WP : (*Local Id: 6 *)
            ACT_SortWP(N);
        END_STEP

        STEP SetAutomaticExecuteCompleted : (*Local Id: 9 *)
        END_STEP
        TRANSITION FROM (LargeSortingConveyor_ACT_AutomaticExecute_Init) TO (Interstep) := (Check_AllowedToOperate AND NOT AutomaticExecuteCompleted AND NOT GVL.IsSFCResetting); END_TRANSITION
        TRANSITION FROM (Interstep) TO (Sort_WP) := (Check_AllowedToOperate AND Interstep.t>T#500ms); END_TRANSITION
        TRANSITION FROM (Sort_WP) TO (SetAutomaticExecuteCompleted) := (WPSorted); END_TRANSITION
        TRANSITION FROM (SetAutomaticExecuteCompleted) TO (LargeSortingConveyor_ACT_AutomaticExecute_Init) := (AutomaticExecuteCompleted); END_TRANSITION
    END_ACTION
    ACTION ACT_EmergencyStop

        INITIAL_STEP Conveyor_ACT_EmergencyStop_Init : (*Local Id: 0 *)
        END_STEP

        STEP ResetVariables : (*Local Id: 3 *)
            Reset_Variables(N);
        END_STEP

        STEP Stop_Conveyor : (*Local Id: 6 *)
            Motor.ACT_Stop(N);
        END_STEP

        STEP Pusher1_Retracting_ES : (*Local Id: 9 *)
            Seperator1.ACT_Retract(N);
        END_STEP

        STEP Pusher2_Retracting_ES : (*Local Id: 12 *)
            Seperator2.ACT_Retract(N);
        END_STEP

        STEP Switch_Retract : (*Local Id: 15 *)
            Switch.ACT_Retract(N);
        END_STEP

        STEP Conveyor_EmergencyHandled : (*Local Id: 18 *)
        END_STEP
        TRANSITION FROM (Conveyor_ACT_EmergencyStop_Init) TO (ResetVariables) := (Not EmergencyHandled AND NOT GVL.IsSFCResetting); END_TRANSITION
        TRANSITION FROM (ResetVariables) TO (Stop_Conveyor) := (NOT InitCompleted AND NOT AutomaticExecuteCompleted); END_TRANSITION
        TRANSITION FROM (Stop_Conveyor) TO (Pusher1_Retracting_ES) := (Motor.Stopped); END_TRANSITION
        TRANSITION FROM (Pusher1_Retracting_ES) TO (Pusher2_Retracting_ES) := (Seperator1.Retracted); END_TRANSITION
        TRANSITION FROM (Pusher2_Retracting_ES) TO (Switch_Retract) := (Seperator2.Retracted); END_TRANSITION
        TRANSITION FROM (Switch_Retract) TO (Conveyor_EmergencyHandled) := (Switch.Retracted); END_TRANSITION
        TRANSITION FROM (Conveyor_EmergencyHandled) TO (Conveyor_ACT_EmergencyStop_Init) := (EmergencyHandled); END_TRANSITION
    END_ACTION
    ACTION ACT_Init

        INITIAL_STEP Conveyor_ACT_Init : (*Local Id: 0 *)
        END_STEP

        STEP ExtendSwitch : (*Local Id: 3 *)
            Switch.ACT_Extend(N);
        END_STEP

        STEP TurnConveyorOn : (*Local Id: 6 *)
            Motor.ACT_TurnClockwise(N);
        END_STEP

        STEP AllowFollowConveyorToInit : (*Local Id: 9 *)
        END_STEP

        STEP Stop_Conveyors : (*Local Id: 14 *)
        END_STEP

        STEP RetractSwitch : (*Local Id: 19 *)
            Switch.ACT_Retract(N);
        END_STEP

        STEP Reset_AllowFollowConveyorToInit : (*Local Id: 22 *)
        END_STEP

        STEP SetInitCompleted : (*Local Id: 27 *)
        END_STEP
        TRANSITION FROM (Conveyor_ACT_Init) TO (ExtendSwitch) := (NOT InitCompleted AND NOT GVL.IsSFCResetting); END_TRANSITION
        TRANSITION FROM (ExtendSwitch) TO (TurnConveyorOn) := (Switch.Extended); END_TRANSITION
        TRANSITION FROM (TurnConveyorOn) TO (AllowFollowConveyorToInit) := (Motor.TurningClockwise); END_TRANSITION
        TRANSITION FROM (AllowFollowConveyorToInit) TO (Stop_Conveyors) := (FollowConveyor_AllowedToInit); END_TRANSITION
        TRANSITION FROM (Stop_Conveyors) TO (RetractSwitch) := (Motor.Stopped); END_TRANSITION
        TRANSITION FROM (RetractSwitch) TO (Reset_AllowFollowConveyorToInit) := (Switch.Retracted); END_TRANSITION
        TRANSITION FROM (Reset_AllowFollowConveyorToInit) TO (SetInitCompleted) := (NOT FollowConveyor_AllowedToInit AND Check_FollowConveyorInitCompleted); END_TRANSITION
        TRANSITION FROM (SetInitCompleted) TO (Conveyor_ACT_Init) := (InitCompleted); END_TRANSITION
    END_ACTION

    Panel();
    ACT_CountWPsAtConveyor();
    StartButton := Panel.StartButton;
    ManuelMode := Panel.ManuelMode;
    AutomaticMode := Panel.AutomaticMode;
    EmergencyStop := Panel.EmergencyStop;
    Check_AllowedToOperate := Main.Check_LargeSortingConveyor_AllowedToOperate;
    Check_FollowConveyorInitCompleted := Main.Check_LargeSortingConveyor_FollowConveyorInitCompleted;
    Check_FollowConveyorAutoamticExecuteCompleted := Main.Check_LargeSortingConveyor_FollowConveyorAutoamticExecuteCompleted;
    Check_EngineStop := MAIN.PPU_EngineStop;
    IF Check_EngineStop THEN
    	Motor.ACT_Stop();
    END_IF
END_FUNCTION_BLOCK

FUNCTION_BLOCK LightGrid

    VAR_INPUT
        Panel : OperationPanelExtended;
    END_VAR

    VAR_OUTPUT
        StartButton : BOOL;
        ManuelMode : BOOL;
        AutomaticMode : BOOL;
        EmergencyStop : BOOL;
    END_VAR

    Panel();
    StartButton := Panel.StartButton;
    ManuelMode := Panel.ManuelMode;
    AutomaticMode := Panel.AutomaticMode;
    EmergencyStop := Panel.EmergencyStop;
END_FUNCTION_BLOCK

FUNCTION_BLOCK MagnetValve

    VAR
        DO_Changeover : BOOL;
    END_VAR

END_FUNCTION_BLOCK

FUNCTION_BLOCK MicroSwitch

    VAR
        DI_SwitchTrue : BOOL;
    END_VAR

END_FUNCTION_BLOCK

FUNCTION_BLOCK MonostableCylinder

    VAR_OUTPUT
        Extended : BOOL;
        Retracted : BOOL;
    END_VAR

    VAR
        DI_Extended : BOOL;
        DI_Retracted : BOOL;
        DO_Extend : BOOL;
        DI_BoundaryPressure : BOOL;
        DI_BoundaryFlowPressure : BOOL;
        AI_PressureSensor : INT;
        AI_FlowPressure : INT;
        AI_PositionTransmitter : INT;
        SFCInit : BOOL;
        SFCReset : BOOL;
    END_VAR
    ACTION ACT_Extend

        INITIAL_STEP Init_ACT_Extend : (*Local Id: 0 *)
        END_STEP

        STEP Extend_Cylinder : (*Local Id: 3 *)
        END_STEP

        STEP SetExtended : (*Local Id: 8 *)
        END_STEP
        TRANSITION FROM (Init_ACT_Extend) TO (Extend_Cylinder) := (NOT Extended AND NOT GVL.IsSFCResetting); END_TRANSITION
        TRANSITION FROM (Extend_Cylinder) TO (SetExtended) := (DI_Extended); END_TRANSITION
        TRANSITION FROM (SetExtended) TO (Init_ACT_Extend) := (Extended); END_TRANSITION
    END_ACTION
    ACTION ACT_Retract

        INITIAL_STEP Init_ACT_Retract : (*Local Id: 0 *)
        END_STEP

        STEP Retract_Cylinder : (*Local Id: 3 *)
        END_STEP

        STEP SetRetacted : (*Local Id: 8 *)
        END_STEP
        TRANSITION FROM (Init_ACT_Retract) TO (Retract_Cylinder) := (NOT Retracted AND NOT GVL.IsSFCResetting); END_TRANSITION
        TRANSITION FROM (Retract_Cylinder) TO (SetRetacted) := (DI_Retracted); END_TRANSITION
        TRANSITION FROM (SetRetacted) TO (Init_ACT_Retract) := (Retracted); END_TRANSITION
    END_ACTION

END_FUNCTION_BLOCK

FUNCTION_BLOCK Motor

    VAR_INPUT
        Stopped : BOOL;
        TurningClockwise : BOOL;
        TurningCounterclockwise : BOOL;
    END_VAR

    VAR_OUTPUT
        AI_Position : UINT;
        AI_Speed : UDINT;
    END_VAR

    VAR
        DO_TurnClockwise : BOOL;
        DO_TurnCounterclockwise : BOOL;
    END_VAR
    ACTION ACT_Stop

        DO_TurnClockwise := FALSE;
        DO_TurnCounterclockwise := FALSE;

        Stopped := TRUE;
        TurningClockwise := FALSE;
        TurningCounterclockwise := FALSE;
    END_ACTION
    ACTION ACT_TurnClockwise

        DO_TurnClockwise := TRUE;
        DO_TurnCounterclockwise := FALSE;

        Stopped := FALSE;
        TurningClockwise := TRUE;
        TurningCounterclockwise := FALSE;
    END_ACTION
    ACTION ACT_TurnCounterclockwise

        DO_TurnClockwise := FALSE;
        DO_TurnCounterclockwise := TRUE;

        Stopped := FALSE;
        TurningClockwise := FALSE;
        TurningCounterclockwise := TRUE;
    END_ACTION

END_FUNCTION_BLOCK

FUNCTION_BLOCK OperationPanel

    VAR_OUTPUT
        EmergencyStop : BOOL;
        StartButton : BOOL;
        ManuelMode : BOOL;
        AutomaticMode : BOOL;
    END_VAR

    VAR
        DI_StartButton : BOOL;
        DI_AutomaticButton : BOOL;
        DI_EmergencyStop : BOOL;
        DO_LampGreen : BOOL;
        DO_LampWhite : BOOL;
    END_VAR
    ACTION ACT_TurnLampGreen_Off

        DO_LampGreen := FALSE;
    END_ACTION
    ACTION ACT_TurnLampGreen_On

        DO_LampGreen := TRUE;
    END_ACTION
    ACTION ACT_TurnLampWhite_Off

        DO_LampWhite:=FALSE;
    END_ACTION
    ACTION ACT_TurnLampWhite_On

        DO_LampWhite:=TRUE;
    END_ACTION

    EmergencyStop := NOT DI_EmergencyStop;
    StartButton := DI_StartButton;
    ManuelMode := NOT DI_AutomaticButton;
    AutomaticMode := DI_AutomaticButton;
END_FUNCTION_BLOCK

FUNCTION_BLOCK OperationPanelExtended

    VAR_OUTPUT
        EmergencyStop : BOOL;
        StartButton : BOOL;
        ManuelMode : BOOL;
        AutomaticMode : BOOL;
        Reset : BOOL;
    END_VAR

    VAR
        DI_EmergencyStop : BOOL;
        DI_StartButton : BOOL;
        DI_AutomaticButton : BOOL;
        DI_StopButton : BOOL;
        DI_ResetButton : BOOL;
        DO_LampGreen : BOOL;
        DO_LampReset : BOOL;
        DO_Q1 : BOOL;
        DO_Q2 : BOOL;
    END_VAR
    ACTION ACT_TurnLampGreen_Off

        DO_LampGreen := FALSE;
    END_ACTION
    ACTION ACT_TurnLampGreen_On

        DO_LampGreen := TRUE;
    END_ACTION
    ACTION ACT_TurnLampReset_Off

        DO_LampReset:=FALSE;
    END_ACTION
    ACTION ACT_TurnLampReset_On

        DO_LampReset:=TRUE;
    END_ACTION

    EmergencyStop := NOT DI_StopButton;
    StartButton := DI_StartButton;
    ManuelMode := NOT DI_AutomaticButton;
    AutomaticMode := DI_AutomaticButton;
    Reset := DI_ResetButton;
END_FUNCTION_BLOCK

FUNCTION_BLOCK OpticalSensor

    VAR
        DI_WPLight : BOOL;
    END_VAR

END_FUNCTION_BLOCK

FUNCTION_BLOCK PicAlpha

    VAR_INPUT
        AtPosition1 : PositionTransmitter;
        AtPosition2 : PositionTransmitter;
        AtPosition3 : PositionTransmitter;
        AtPosition4 : PositionTransmitter;
        Motor : Motor;
        Gripper : VacuumGripperExtended;
        LiftingCylinder : MonostableCylinder;
        SoftwareEmergency : BOOL;
        Check_AllowedToOperate : BOOL;
        Check_Conveyor_AutomaticExecuteCompleted : BOOL;
        Check_EngineStop : BOOL;
        SFCReset : BOOL;
    END_VAR

    VAR_OUTPUT
        InitCompleted : BOOL;
        Conveyor_AllowedToOperate : BOOL;
        AutomaticExecuteCompleted : BOOL;
        EmergencyHandled : BOOL;
    END_VAR

    VAR
        WPPickedUp : BOOL;
        WPPutDown : BOOL;
        ReachedPosition1 : BOOL;
        ReachedPosition2 : BOOL;
        ReachedPosition3 : BOOL;
        ReachedPosition4 : BOOL;
        SFCInit : BOOL;
    END_VAR
    ACTION Reset_Variables

        InitCompleted := FALSE;
        Conveyor_AllowedToOperate := FALSE;
        AutomaticExecuteCompleted := FALSE;

        WPPickedUp := FALSE;
        WPPutDown := FALSE;
        ReachedPosition1 := FALSE;
        ReachedPosition2 := FALSE;
        ReachedPosition3 := FALSE;
        ReachedPosition4 := FALSE;
    END_ACTION
    ACTION ACT_MoveToPos1

        INITIAL_STEP Init_ACT_MoveToPos1 : (*Local Id: 0 *)
        END_STEP

        STEP DecideHowToMove_Pos1 : (*Local Id: 3 *)
        END_STEP

        STEP Turn_Backwards : (*Local Id: 7 *)
            Motor.ACT_TurnCounterclockwise(N);
        END_STEP

        STEP Turn_Backwards_Pos1 : (*Local Id: 12 *)
            Motor.ACT_TurnCounterclockwise(N);
        END_STEP

        STEP Turn_Forwards_Pos1 : (*Local Id: 18 *)
            Motor.ACT_TurnClockwise(N);
        END_STEP

        STEP Stop_Motor_Pos1 : (*Local Id: 23 *)
            Motor.ACT_Stop(N);
        END_STEP

        STEP Position1_Reached : (*Local Id: 26 *)
        END_STEP
        TRANSITION FROM (DecideHowToMove_Pos1) TO (Turn_Backwards) := (AtPosition2.DI_PositionReached OR AtPosition3.DI_PositionReached OR AtPosition4.DI_PositionReached); END_TRANSITION
        TRANSITION FROM (DecideHowToMove_Pos1) TO (Turn_Backwards_Pos1) := (NOT (AtPosition2.DI_PositionReached AND AtPosition3.DI_PositionReached AND AtPosition4.DI_PositionReached)); END_TRANSITION
        TRANSITION FROM (Turn_Backwards_Pos1) TO (Stop_Motor_Pos1) := (AtPosition1.DI_PositionReached); END_TRANSITION
        TRANSITION FROM (Turn_Backwards_Pos1) TO (Turn_Forwards_Pos1) := (NOT AtPosition1.DI_PositionReached AND Turn_Backwards_Pos1.t>T#4s); END_TRANSITION
        TRANSITION FROM (Turn_Backwards_Pos1) TO (Stop_Motor_Pos1) := (AtPosition1.DI_PositionReached); END_TRANSITION
        TRANSITION FROM (Turn_Forwards_Pos1) TO (Stop_Motor_Pos1) := (AtPosition1.DI_PositionReached); END_TRANSITION
        TRANSITION FROM (Turn_Backwards) TO (Stop_Motor_Pos1) := (AtPosition1.DI_PositionReached); END_TRANSITION
        TRANSITION FROM (Turn_Backwards_Pos1) TO (Stop_Motor_Pos1) := (AtPosition1.DI_PositionReached); END_TRANSITION
        TRANSITION FROM (Turn_Forwards_Pos1) TO (Stop_Motor_Pos1) := (AtPosition1.DI_PositionReached); END_TRANSITION
        TRANSITION FROM (Init_ACT_MoveToPos1) TO (DecideHowToMove_Pos1) := (NOT ReachedPosition1 AND NOT GVL.IsSFCResetting); END_TRANSITION
        TRANSITION FROM (Stop_Motor_Pos1) TO (Position1_Reached) := (Motor.Stopped); END_TRANSITION
        TRANSITION FROM (Position1_Reached) TO (Init_ACT_MoveToPos1) := (ReachedPosition1); END_TRANSITION
    END_ACTION
    ACTION ACT_MoveToPos2

        INITIAL_STEP Init_ACT_MoveToPos2 : (*Local Id: 0 *)
        END_STEP

        STEP DecideHowToMove_Pos2 : (*Local Id: 3 *)
        END_STEP

        STEP Move_Forwards : (*Local Id: 7 *)
            Motor.ACT_TurnClockwise(N);
        END_STEP

        STEP Move_Backwards : (*Local Id: 12 *)
            Motor.ACT_TurnCounterclockwise(N);
        END_STEP

        STEP Turn_Backwards_Pos2 : (*Local Id: 17 *)
            Motor.ACT_TurnCounterclockwise(N);
        END_STEP

        STEP Turn_Forwards_Pos2 : (*Local Id: 23 *)
            Motor.ACT_TurnClockwise(N);
        END_STEP

        STEP Stop_Motor_Pos2 : (*Local Id: 28 *)
            Motor.ACT_Stop(N);
        END_STEP

        STEP Position2_Reached : (*Local Id: 31 *)
        END_STEP
        TRANSITION FROM (DecideHowToMove_Pos2) TO (Move_Forwards) := (AtPosition1.DI_PositionReached); END_TRANSITION
        TRANSITION FROM (DecideHowToMove_Pos2) TO (Move_Backwards) := (AtPosition3.DI_PositionReached OR AtPosition4.DI_PositionReached); END_TRANSITION
        TRANSITION FROM (DecideHowToMove_Pos2) TO (Turn_Backwards_Pos2) := (NOT (AtPosition1.DI_PositionReached AND AtPosition3.DI_PositionReached AND AtPosition4.DI_PositionReached)); END_TRANSITION
        TRANSITION FROM (Turn_Backwards_Pos2) TO (Stop_Motor_Pos2) := (AtPosition2.DI_PositionReached); END_TRANSITION
        TRANSITION FROM (Turn_Backwards_Pos2) TO (Turn_Forwards_Pos2) := (NOT AtPosition2.DI_PositionReached AND Turn_Backwards_Pos2.t>T#4s); END_TRANSITION
        TRANSITION FROM (Turn_Backwards_Pos2) TO (Stop_Motor_Pos2) := (AtPosition2.DI_PositionReached); END_TRANSITION
        TRANSITION FROM (Turn_Forwards_Pos2) TO (Stop_Motor_Pos2) := (AtPosition2.DI_PositionReached); END_TRANSITION
        TRANSITION FROM (Move_Forwards) TO (Stop_Motor_Pos2) := (AtPosition2.DI_PositionReached); END_TRANSITION
        TRANSITION FROM (Move_Backwards) TO (Stop_Motor_Pos2) := (AtPosition2.DI_PositionReached); END_TRANSITION
        TRANSITION FROM (Turn_Backwards_Pos2) TO (Stop_Motor_Pos2) := (AtPosition2.DI_PositionReached); END_TRANSITION
        TRANSITION FROM (Turn_Forwards_Pos2) TO (Stop_Motor_Pos2) := (AtPosition2.DI_PositionReached); END_TRANSITION
        TRANSITION FROM (Init_ACT_MoveToPos2) TO (DecideHowToMove_Pos2) := (NOT ReachedPosition2 AND NOT GVL.IsSFCResetting); END_TRANSITION
        TRANSITION FROM (Stop_Motor_Pos2) TO (Position2_Reached) := (Motor.Stopped); END_TRANSITION
        TRANSITION FROM (Position2_Reached) TO (Init_ACT_MoveToPos2) := (ReachedPosition2); END_TRANSITION
    END_ACTION
    ACTION ACT_MoveToPos3

        INITIAL_STEP Init_ACT_MoveToPos3 : (*Local Id: 0 *)
        END_STEP

        STEP DecideHowToMove_Pos3 : (*Local Id: 3 *)
        END_STEP

        STEP Move_Forwards : (*Local Id: 7 *)
            Motor.ACT_TurnClockwise(N);
        END_STEP

        STEP Move_Backwards : (*Local Id: 12 *)
            Motor.ACT_TurnCounterclockwise(N);
        END_STEP

        STEP Move_Backwards_Pos3 : (*Local Id: 17 *)
            Motor.ACT_TurnCounterclockwise(N);
        END_STEP

        STEP Move_Forwards__Pos3 : (*Local Id: 23 *)
            Motor.ACT_TurnClockwise(N);
        END_STEP

        STEP Stop_Motor_Pos3 : (*Local Id: 28 *)
            Motor.ACT_Stop(N);
        END_STEP

        STEP Position3_Reached : (*Local Id: 31 *)
        END_STEP
        TRANSITION FROM (DecideHowToMove_Pos3) TO (Move_Forwards) := (AtPosition1.DI_PositionReached OR AtPosition2.DI_PositionReached); END_TRANSITION
        TRANSITION FROM (DecideHowToMove_Pos3) TO (Move_Backwards) := (AtPosition4.DI_PositionReached); END_TRANSITION
        TRANSITION FROM (DecideHowToMove_Pos3) TO (Move_Backwards_Pos3) := (NOT(AtPosition1.DI_PositionReached AND AtPosition2.DI_PositionReached AND AtPosition4.DI_PositionReached)); END_TRANSITION
        TRANSITION FROM (Move_Backwards_Pos3) TO (Stop_Motor_Pos3) := (AtPosition3.DI_PositionReached); END_TRANSITION
        TRANSITION FROM (Move_Backwards_Pos3) TO (Move_Forwards__Pos3) := (NOT AtPosition3.DI_PositionReached AND Move_Backwards_Pos3.t>T#4s); END_TRANSITION
        TRANSITION FROM (Move_Backwards_Pos3) TO (Stop_Motor_Pos3) := (AtPosition3.DI_PositionReached); END_TRANSITION
        TRANSITION FROM (Move_Forwards__Pos3) TO (Stop_Motor_Pos3) := (AtPosition3.DI_PositionReached); END_TRANSITION
        TRANSITION FROM (Move_Forwards) TO (Stop_Motor_Pos3) := (AtPosition3.DI_PositionReached); END_TRANSITION
        TRANSITION FROM (Move_Backwards) TO (Stop_Motor_Pos3) := (AtPosition3.DI_PositionReached); END_TRANSITION
        TRANSITION FROM (Move_Backwards_Pos3) TO (Stop_Motor_Pos3) := (AtPosition3.DI_PositionReached); END_TRANSITION
        TRANSITION FROM (Move_Forwards__Pos3) TO (Stop_Motor_Pos3) := (AtPosition3.DI_PositionReached); END_TRANSITION
        TRANSITION FROM (Init_ACT_MoveToPos3) TO (DecideHowToMove_Pos3) := (NOT ReachedPosition3 AND NOT GVL.IsSFCResetting); END_TRANSITION
        TRANSITION FROM (Stop_Motor_Pos3) TO (Position3_Reached) := (Motor.Stopped); END_TRANSITION
        TRANSITION FROM (Position3_Reached) TO (Init_ACT_MoveToPos3) := (ReachedPosition3); END_TRANSITION
    END_ACTION
    ACTION ACT_MoveToPos4

        INITIAL_STEP Init_ACT_MoveToPos4 : (*Local Id: 0 *)
        END_STEP

        STEP DecideHowToMove_Pos4 : (*Local Id: 3 *)
        END_STEP

        STEP Move_Forwards : (*Local Id: 7 *)
            Motor.ACT_TurnClockwise(N);
        END_STEP

        STEP Move_Backwards_Pos4 : (*Local Id: 12 *)
            Motor.ACT_TurnCounterclockwise(N);
        END_STEP

        STEP Move_Forwards_Pos4 : (*Local Id: 18 *)
            Motor.ACT_TurnClockwise(N);
        END_STEP

        STEP Stop_Motor_Pos4 : (*Local Id: 23 *)
            Motor.ACT_Stop(N);
        END_STEP

        STEP Position4_Reached : (*Local Id: 26 *)
        END_STEP
        TRANSITION FROM (DecideHowToMove_Pos4) TO (Move_Forwards) := (AtPosition1.DI_PositionReached OR AtPosition2.DI_PositionReached OR AtPosition3.DI_PositionReached); END_TRANSITION
        TRANSITION FROM (DecideHowToMove_Pos4) TO (Move_Backwards_Pos4) := (NOT(AtPosition1.DI_PositionReached AND AtPosition2.DI_PositionReached AND AtPosition3.DI_PositionReached)); END_TRANSITION
        TRANSITION FROM (Move_Backwards_Pos4) TO (Stop_Motor_Pos4) := (AtPosition4.DI_PositionReached); END_TRANSITION
        TRANSITION FROM (Move_Backwards_Pos4) TO (Move_Forwards_Pos4) := (NOT AtPosition4.DI_PositionReached AND Move_Backwards_Pos4.t>T#4s); END_TRANSITION
        TRANSITION FROM (Move_Backwards_Pos4) TO (Stop_Motor_Pos4) := (AtPosition4.DI_PositionReached); END_TRANSITION
        TRANSITION FROM (Move_Forwards_Pos4) TO (Stop_Motor_Pos4) := (AtPosition4.DI_PositionReached); END_TRANSITION
        TRANSITION FROM (Move_Forwards) TO (Stop_Motor_Pos4) := (AtPosition4.DI_PositionReached); END_TRANSITION
        TRANSITION FROM (Move_Backwards_Pos4) TO (Stop_Motor_Pos4) := (AtPosition4.DI_PositionReached); END_TRANSITION
        TRANSITION FROM (Move_Forwards_Pos4) TO (Stop_Motor_Pos4) := (AtPosition4.DI_PositionReached); END_TRANSITION
        TRANSITION FROM (Init_ACT_MoveToPos4) TO (DecideHowToMove_Pos4) := (NOT ReachedPosition4 AND NOT GVL.IsSFCResetting); END_TRANSITION
        TRANSITION FROM (Stop_Motor_Pos4) TO (Position4_Reached) := (Motor.Stopped); END_TRANSITION
        TRANSITION FROM (Position4_Reached) TO (Init_ACT_MoveToPos4) := (ReachedPosition4); END_TRANSITION
    END_ACTION
    ACTION ACT_PickUpWP

        INITIAL_STEP Init_ACT_PickUpWP : (*Local Id: 0 *)
        END_STEP

        STEP PicAlpha_Down : (*Local Id: 3 *)
            LiftingCylinder.ACT_Extend(N);
        END_STEP

        STEP Turn_VacuumOn : (*Local Id: 6 *)
            Gripper.ACT_Intake(N);
        END_STEP

        STEP PicAlpha_Up : (*Local Id: 10 *)
            LiftingCylinder.ACT_Retract(N);
        END_STEP

        STEP WP_PickedUp : (*Local Id: 13 *)
        END_STEP

        STEP Error : (*Local Id: 20 *)
        END_STEP
        TRANSITION FROM (Turn_VacuumOn) TO (PicAlpha_Up) := (Gripper.Intaken); END_TRANSITION
        TRANSITION FROM (Turn_VacuumOn) TO (Error) := (Turn_VacuumOn.t>T#2s AND NOT Gripper.Intaken); END_TRANSITION
        TRANSITION FROM (WP_PickedUp) TO (Init_ACT_PickUpWP) := (WPPickedUp); END_TRANSITION
        TRANSITION FROM (Error) TO (Init_ACT_PickUpWP) := (SoftwareEmergency); END_TRANSITION
        TRANSITION FROM (Init_ACT_PickUpWP) TO (PicAlpha_Down) := (NOT GVL.IsSFCResetting); END_TRANSITION
        TRANSITION FROM (PicAlpha_Down) TO (Turn_VacuumOn) := (LiftingCylinder.Extended); END_TRANSITION
        TRANSITION FROM (PicAlpha_Up) TO (WP_PickedUp) := (LiftingCylinder.Retracted); END_TRANSITION
    END_ACTION
    ACTION ACT_PutDownWP

        INITIAL_STEP Init_ACT_PutDownWP : (*Local Id: 0 *)
        END_STEP

        STEP PicAlpha_Down : (*Local Id: 3 *)
            LiftingCylinder.ACT_Extend(N);
        END_STEP

        STEP Releasing_WP : (*Local Id: 6 *)
            Gripper.ACT_Release(N);
        END_STEP

        STEP PicAlpha_Up : (*Local Id: 9 *)
            LiftingCylinder.ACT_Retract(N);
        END_STEP

        STEP WP_PutDown : (*Local Id: 12 *)
        END_STEP
        TRANSITION FROM (Init_ACT_PutDownWP) TO (PicAlpha_Down) := (NOT GVL.IsSFCResetting); END_TRANSITION
        TRANSITION FROM (PicAlpha_Down) TO (Releasing_WP) := (LiftingCylinder.Extended); END_TRANSITION
        TRANSITION FROM (Releasing_WP) TO (PicAlpha_Up) := (Gripper.Released); END_TRANSITION
        TRANSITION FROM (PicAlpha_Up) TO (WP_PutDown) := (LiftingCylinder.Retracted); END_TRANSITION
        TRANSITION FROM (WP_PutDown) TO (Init_ACT_PutDownWP) := (WPPutDown); END_TRANSITION
    END_ACTION
    ACTION ACT_AutomaticExecute

        INITIAL_STEP Init_ACT_AutomaticExecute : (*Local Id: 0 *)
        END_STEP

        STEP Interstep : (*Local Id: 3 *)
        END_STEP

        STEP Move_To_Pos1 : (*Local Id: 6 *)
            ACT_MoveToPos1(N);
        END_STEP

        STEP PickUpWP : (*Local Id: 9 *)
            ACT_PickUpWP(N);
        END_STEP

        STEP Move_To_Pos3 : (*Local Id: 12 *)
            ACT_MoveToPos3(N);
        END_STEP

        STEP PutDownWP : (*Local Id: 15 *)
            ACT_PutDownWP(N);
        END_STEP

        STEP SetAutomaticExecuteCompleted : (*Local Id: 18 *)
        END_STEP
        TRANSITION FROM (Init_ACT_AutomaticExecute) TO (Interstep) := (Check_AllowedToOperate AND NOT AutomaticExecuteCompleted AND NOT GVL.IsSFCResetting); END_TRANSITION
        TRANSITION FROM (Interstep) TO (Move_To_Pos1) := (Check_AllowedToOperate AND Interstep.t>T#500ms); END_TRANSITION
        TRANSITION FROM (Move_To_Pos1) TO (PickUpWP) := (ReachedPosition1); END_TRANSITION
        TRANSITION FROM (PickUpWP) TO (Move_To_Pos3) := (WPPickedUp); END_TRANSITION
        TRANSITION FROM (Move_To_Pos3) TO (PutDownWP) := (ReachedPosition3); END_TRANSITION
        TRANSITION FROM (PutDownWP) TO (SetAutomaticExecuteCompleted) := (WPPutDown); END_TRANSITION
        TRANSITION FROM (SetAutomaticExecuteCompleted) TO (Init_ACT_AutomaticExecute) := (AutomaticExecuteCompleted); END_TRANSITION
    END_ACTION
    ACTION ACT_EmergencyStop

        INITIAL_STEP Init_ACT_EmergencyStop : (*Local Id: 0 *)
        END_STEP

        STEP ResetVariables : (*Local Id: 3 *)
            Reset_Variables(N);
        END_STEP

        STEP StopPicAlpha : (*Local Id: 6 *)
            Motor.ACT_Stop(N);
        END_STEP

        STEP Turn_Vacuum_Off : (*Local Id: 12 *)
            Gripper.ACT_Release(N);
        END_STEP

        STEP Retract_LiftingCylinder : (*Local Id: 16 *)
            LiftingCylinder.ACT_Retract(N);
        END_STEP

        STEP PicAlpha_EmergencyHandled : (*Local Id: 19 *)
        END_STEP
        TRANSITION FROM (StopPicAlpha) TO (Retract_LiftingCylinder) := (Motor.Stopped AND Gripper.Intaken); END_TRANSITION
        TRANSITION FROM (StopPicAlpha) TO (Turn_Vacuum_Off) := (Motor.Stopped AND NOT Gripper.Intaken); END_TRANSITION
        TRANSITION FROM (StopPicAlpha) TO (Retract_LiftingCylinder) := (Motor.Stopped AND Gripper.Intaken); END_TRANSITION
        TRANSITION FROM (Turn_Vacuum_Off) TO (Retract_LiftingCylinder) := (Gripper.Released); END_TRANSITION
        TRANSITION FROM (Init_ACT_EmergencyStop) TO (ResetVariables) := (NOT EmergencyHandled AND NOT GVL.IsSFCResetting); END_TRANSITION
        TRANSITION FROM (ResetVariables) TO (StopPicAlpha) := (NOT InitCompleted AND NOT AutomaticExecuteCompleted); END_TRANSITION
        TRANSITION FROM (Retract_LiftingCylinder) TO (PicAlpha_EmergencyHandled) := (LiftingCylinder.Retracted); END_TRANSITION
        TRANSITION FROM (PicAlpha_EmergencyHandled) TO (Init_ACT_EmergencyStop) := (EmergencyHandled); END_TRANSITION
    END_ACTION
    ACTION ACT_Init

        INITIAL_STEP Init_ACT_Init : (*Local Id: 0 *)
        END_STEP

        STEP Move_Up : (*Local Id: 3 *)
            LiftingCylinder.ACT_Retract(N);
        END_STEP

        STEP WPAllreadyPickedUp : (*Local Id: 9 *)
        END_STEP

        STEP Move_ToPos3 : (*Local Id: 14 *)
            ACT_MoveToPos3(N);
        END_STEP

        STEP Put_WP_On_Conveyor : (*Local Id: 17 *)
            ACT_PutDownWP(N);
        END_STEP

        STEP SetInitCompleted : (*Local Id: 21 *)
        END_STEP
        TRANSITION FROM (Move_Up) TO (SetInitCompleted) := (LiftingCylinder.Retracted AND NOT Gripper.VacuumSwitch.DI_TakenIn); END_TRANSITION
        TRANSITION FROM (Move_Up) TO (WPAllreadyPickedUp) := (LiftingCylinder.Retracted AND Gripper.VacuumSwitch.DI_TakenIn); END_TRANSITION
        TRANSITION FROM (Move_Up) TO (SetInitCompleted) := (LiftingCylinder.Retracted AND NOT Gripper.VacuumSwitch.DI_TakenIn); END_TRANSITION
        TRANSITION FROM (Put_WP_On_Conveyor) TO (SetInitCompleted) := (WPPutDown); END_TRANSITION
        TRANSITION FROM (Init_ACT_Init) TO (Move_Up) := (NOT InitCompleted AND NOT GVL.IsSFCResetting); END_TRANSITION
        TRANSITION FROM (WPAllreadyPickedUp) TO (Move_ToPos3) := (WPPickedUp); END_TRANSITION
        TRANSITION FROM (Move_ToPos3) TO (Put_WP_On_Conveyor) := (ReachedPosition3); END_TRANSITION
        TRANSITION FROM (SetInitCompleted) TO (Init_ACT_Init) := (InitCompleted); END_TRANSITION
    END_ACTION

    Check_AllowedToOperate := MAIN.Check_PicAlpha_AllowedToOperate;
    Check_Conveyor_AutomaticExecuteCompleted := MAIN.Check_PicAlpha_Conveyor_AutomaticExecuteCompleted;
    Check_EngineStop := MAIN.PPU_EngineStop;
    IF Check_EngineStop THEN
    	Motor.ACT_Stop();
    END_IF
END_FUNCTION_BLOCK

FUNCTION_BLOCK PicAlphaConveyor

    VAR_INPUT
        PsSwitch : PresenceSensor;
        PsEnd : PresenceSensor;
        Switch : Switch;
        Motor : Motor;
        Check_AllowedToInit : BOOL;
        Check_AllowedToReceive : BOOL;
        Check_AllowedToSend : BOOL;
        Check_FollowConveyor_InitCompleted : BOOL;
        Check_PicAlpha_AutomaticExecuteCompleted : BOOL;
        Check_FollowConveyor_AutomaticExecuteCompleted : BOOL;
        Check_EngineStop : BOOL;
        SFCReset : BOOL;
    END_VAR

    VAR_OUTPUT
        InitCompleted : BOOL;
        FollowConveyor_AllowedToInit : BOOL;
        PicAlpha_AllowedToOperate : BOOL;
        FollowConveyor_AllowedToOperate : BOOL;
        AutomaticExecuteReceivingCompleted : BOOL;
        AutomaticExecuteSendingCompleted : BOOL;
        EmergencyHandled : BOOL;
    END_VAR

    VAR
        ConveyorSpeed : INT;
        NumberOfWPs : INT;
        WPSeperated : BOOL;
        SFCInit : BOOL;
    END_VAR
    ACTION Reduce_WPNumber

        NumberOfWPs := NumberOfWPs-1;
    END_ACTION
    ACTION Reset_FollowConveyorAllowedToInit

        FollowConveyor_AllowedToInit := FALSE;
    END_ACTION
    ACTION Reset_FollowConveyorAllowedToOperate

        FollowConveyor_AllowedToOperate := FALSE;
    END_ACTION
    ACTION Reset_Variables

        InitCompleted := FALSE;
        FollowConveyor_AllowedToInit := FALSE;
        PicAlpha_AllowedToOperate := FALSE;
        FollowConveyor_AllowedToOperate := FALSE;
        AutomaticExecuteReceivingCompleted := FALSE;
        AutomaticExecuteSendingCompleted := FALSE;

        NumberOfWPs := 0;
        WPSeperated := FALSE;
    END_ACTION
    ACTION Rest_PicAlpha_AllowedToOperate

        PicAlpha_AllowedToOperate := FALSE;
    END_ACTION
    ACTION Set_FollowConveyorAllowedToInit

        FollowConveyor_AllowedToInit := TRUE;
    END_ACTION
    ACTION Set_FollowConveyorAllowedToOperate

        FollowConveyor_AllowedToOperate := TRUE;
    END_ACTION
    ACTION Set_NumberOfWPsTo3

        NumberOfWPs := 3;
    END_ACTION
    ACTION Set_PicAlpha_AllowedToOperate

        PicAlpha_AllowedToOperate := TRUE;
    END_ACTION
    ACTION ACT_SeperateWP

        INITIAL_STEP Init_ACT_SeperateWP : (*Local Id: 0 *)
        END_STEP

        STEP ExtendSwitch : (*Local Id: 3 *)
            Switch.ACT_Extend(N);
        END_STEP

        STEP RetractSwitch : (*Local Id: 6 *)
            Switch.ACT_Retract(N);
        END_STEP

        STEP WP_Seperated : (*Local Id: 9 *)
        END_STEP
        TRANSITION FROM (Init_ACT_SeperateWP) TO (ExtendSwitch) := (NOT WPSeperated AND NOT GVL.IsSFCResetting); END_TRANSITION
        TRANSITION FROM (ExtendSwitch) TO (RetractSwitch) := (Switch.Extended); END_TRANSITION
        TRANSITION FROM (RetractSwitch) TO (WP_Seperated) := (Switch.Retracted); END_TRANSITION
        TRANSITION FROM (WP_Seperated) TO (Init_ACT_SeperateWP) := (WPSeperated); END_TRANSITION
    END_ACTION
    ACTION ACT_AutomaticExecute

        INITIAL_STEP Init_ACT_AutomaticExecute : (*Local Id: 0 *)
        END_STEP

        STEP Choice_ReceivingSending : (*Local Id: 3 *)
        END_STEP

        STEP Interstep_Receiving : (*Local Id: 7 *)
        END_STEP

        STEP ConveyorForwards_Receiving : (*Local Id: 15 *)
            Motor.ACT_TurnClockwise(N);
        END_STEP

        STEP StopConveyor_Receiving : (*Local Id: 18 *)
        END_STEP

        STEP ReceivingCompleted : (*Local Id: 23 *)
        END_STEP

        STEP Interstep_Sending : (*Local Id: 30 *)
        END_STEP

        STEP ThreeWPsAvailable : (*Local Id: 38 *)
            Set_NumberOfWPsTo3(N);
        END_STEP

        STEP PicAlphaOperating : (*Local Id: 41 *)
            Set_PicAlpha_AllowedToOperate(P0);
            Rest_PicAlpha_AllowedToOperate(P1);
        END_STEP

        STEP ConveyorForwards_Sending : (*Local Id: 44 *)
            Motor.ACT_TurnClockwise(N);
        END_STEP

        STEP SortWP_fromPicAlpha : (*Local Id: 47 *)
            Set_FollowConveyorAllowedToOperate(P0);
            Reset_FollowConveyorAllowedToOperate(P1);
        END_STEP

        STEP ReduceWPNumber : (*Local Id: 50 *)
            Reduce_WPNumber(N);
        END_STEP

        STEP ConveyorForwards_Sending_again : (*Local Id: 53 *)
            Motor.ACT_TurnClockwise(N);
        END_STEP

        STEP SeperateWP : (*Local Id: 56 *)
            ACT_SeperateWP(N);
        END_STEP

        STEP StopConveyor_Sending : (*Local Id: 59 *)
        END_STEP

        STEP SortWP : (*Local Id: 64 *)
            Set_FollowConveyorAllowedToOperate(P0);
            Reset_FollowConveyorAllowedToOperate(P1);
        END_STEP

        STEP ReduceWPNumber_again : (*Local Id: 67 *)
            Reduce_WPNumber(N);
        END_STEP
        TRANSITION FROM (Choice_ReceivingSending) TO (Interstep_Receiving) := (Check_AllowedToReceive); END_TRANSITION
        TRANSITION FROM (Choice_ReceivingSending) TO (Interstep_Sending) := (Check_AllowedToSend); END_TRANSITION
        TRANSITION FROM (Interstep_Receiving) TO (ConveyorForwards_Receiving) := (Check_AllowedToReceive AND Interstep_Receiving.t>T#100ms); END_TRANSITION
        TRANSITION FROM (Interstep_Receiving) TO (Init_ACT_AutomaticExecute) := (NOT Check_AllowedToReceive AND Interstep_Receiving.t>T#100ms); END_TRANSITION
        TRANSITION FROM (Interstep_Sending) TO (ThreeWPsAvailable) := (Check_AllowedToSend AND Interstep_Sending.t>T#100ms); END_TRANSITION
        TRANSITION FROM (Interstep_Sending) TO (Init_ACT_AutomaticExecute) := (NOT Check_AllowedToSend AND Interstep_Sending.t>T#100ms); END_TRANSITION
        TRANSITION FROM (ReduceWPNumber_again) TO (Init_ACT_AutomaticExecute) := (NumberOfWPs<=0); END_TRANSITION
        TRANSITION FROM (ReduceWPNumber_again) TO (ConveyorForwards_Sending_again) := (NumberOfWPs>0); END_TRANSITION
        TRANSITION FROM (Interstep_Receiving) TO (ConveyorForwards_Receiving) := (Check_AllowedToReceive AND Interstep_Receiving.t>T#100ms); END_TRANSITION
        TRANSITION FROM (Interstep_Sending) TO (ThreeWPsAvailable) := (Check_AllowedToSend AND Interstep_Sending.t>T#100ms); END_TRANSITION
        TRANSITION FROM (ReduceWPNumber_again) TO (Init_ACT_AutomaticExecute) := (NumberOfWPs<=0); END_TRANSITION
        TRANSITION FROM (ReceivingCompleted) TO (Init_ACT_AutomaticExecute) := (AutomaticExecuteReceivingCompleted); END_TRANSITION
        TRANSITION FROM (ReduceWPNumber_again) TO (Init_ACT_AutomaticExecute) := (NumberOfWPs<=0); END_TRANSITION
        TRANSITION FROM (Init_ACT_AutomaticExecute) TO (Choice_ReceivingSending) := (NOT AutomaticExecuteReceivingCompleted AND NOT AutomaticExecuteSendingCompleted AND NOT GVL.IsSFCResetting); END_TRANSITION
        TRANSITION FROM (ConveyorForwards_Receiving) TO (StopConveyor_Receiving) := (Motor.TurningClockwise); END_TRANSITION
        TRANSITION FROM (StopConveyor_Receiving) TO (ReceivingCompleted) := (Motor.Stopped); END_TRANSITION
        TRANSITION FROM (ThreeWPsAvailable) TO (PicAlphaOperating) := (NumberOfWPs=3); END_TRANSITION
        TRANSITION FROM (PicAlphaOperating) TO (ConveyorForwards_Sending) := (Check_PicAlpha_AutomaticExecuteCompleted); END_TRANSITION
        TRANSITION FROM (ConveyorForwards_Sending) TO (SortWP_fromPicAlpha) := (Motor.TurningClockwise); END_TRANSITION
        TRANSITION FROM (SortWP_fromPicAlpha) TO (ReduceWPNumber) := (Check_FollowConveyor_AutomaticExecuteCompleted); END_TRANSITION
        TRANSITION FROM (ReduceWPNumber) TO (ConveyorForwards_Sending_again) := (NumberOfWPs=2); END_TRANSITION
        TRANSITION FROM (ConveyorForwards_Sending_again) TO (SeperateWP) := (Motor.TurningClockwise); END_TRANSITION
        TRANSITION FROM (SeperateWP) TO (StopConveyor_Sending) := (WPSeperated); END_TRANSITION
        TRANSITION FROM (StopConveyor_Sending) TO (SortWP) := (Motor.Stopped); END_TRANSITION
        TRANSITION FROM (SortWP) TO (ReduceWPNumber_again) := (Check_FollowConveyor_AutomaticExecuteCompleted); END_TRANSITION
    END_ACTION
    ACTION ACT_EmergencyStop

        INITIAL_STEP Init_ACT_EmergencyStop : (*Local Id: 0 *)
        END_STEP

        STEP ResetVariables : (*Local Id: 3 *)
            Reset_Variables(N);
        END_STEP

        STEP StopConveyor : (*Local Id: 6 *)
            Motor.ACT_Stop(N);
        END_STEP

        STEP RetractSwitch : (*Local Id: 9 *)
            Switch.ACT_Retract(N);
        END_STEP

        STEP PicAlphaConveyor_EmergencyHandled : (*Local Id: 12 *)
        END_STEP
        TRANSITION FROM (Init_ACT_EmergencyStop) TO (ResetVariables) := (NOT EmergencyHandled AND NOT GVL.IsSFCResetting); END_TRANSITION
        TRANSITION FROM (ResetVariables) TO (StopConveyor) := (NOT InitCompleted AND NOT AutomaticExecuteReceivingCompleted); END_TRANSITION
        TRANSITION FROM (StopConveyor) TO (RetractSwitch) := (Motor.Stopped); END_TRANSITION
        TRANSITION FROM (RetractSwitch) TO (PicAlphaConveyor_EmergencyHandled) := (Switch.Retracted); END_TRANSITION
        TRANSITION FROM (PicAlphaConveyor_EmergencyHandled) TO (Init_ACT_EmergencyStop) := (EmergencyHandled); END_TRANSITION
    END_ACTION
    ACTION ACT_Init

        INITIAL_STEP Init_ACT_Init : (*Local Id: 0 *)
        END_STEP

        STEP Interstep : (*Local Id: 5 *)
        END_STEP

        STEP RetractSwitch : (*Local Id: 13 *)
            Switch.ACT_Retract(N);
        END_STEP

        STEP Wait : (*Local Id: 16 *)
        END_STEP

        STEP ConveyorForwards : (*Local Id: 19 *)
            Motor.ACT_TurnClockwise(N);
        END_STEP

        STEP StopConveyor : (*Local Id: 22 *)
        END_STEP

        STEP AllowFollowConveyor_ToInitialise : (*Local Id: 27 *)
            Set_FollowConveyorAllowedToInit(P0);
            Reset_FollowConveyorAllowedToInit(P1);
        END_STEP

        STEP Init_Completed : (*Local Id: 30 *)
        END_STEP
        TRANSITION FROM (Interstep) TO (RetractSwitch) := (Check_AllowedToInit AND NOT InitCompleted AND Interstep.t>T#500ms); END_TRANSITION
        TRANSITION FROM (Interstep) TO (Init_ACT_Init) := ((NOT Check_AllowedToInit OR InitCompleted) AND Interstep.t>T#500ms); END_TRANSITION
        TRANSITION FROM (Interstep) TO (RetractSwitch) := (Check_AllowedToInit AND NOT InitCompleted AND Interstep.t>T#500ms); END_TRANSITION
        TRANSITION FROM (Init_ACT_Init) TO (Interstep) := (Check_AllowedToInit AND NOT InitCompleted AND NOT GVL.IsSFCResetting); END_TRANSITION
        TRANSITION FROM (RetractSwitch) TO (Wait) := (Switch.Retracted); END_TRANSITION
        TRANSITION FROM (Wait) TO (ConveyorForwards) := (Wait.t>T#2s); END_TRANSITION
        TRANSITION FROM (ConveyorForwards) TO (StopConveyor) := (Motor.TurningClockwise); END_TRANSITION
        TRANSITION FROM (StopConveyor) TO (AllowFollowConveyor_ToInitialise) := (Motor.Stopped); END_TRANSITION
        TRANSITION FROM (AllowFollowConveyor_ToInitialise) TO (Init_Completed) := (Check_FollowConveyor_InitCompleted); END_TRANSITION
        TRANSITION FROM (Init_Completed) TO (Init_ACT_Init) := (InitCompleted); END_TRANSITION
    END_ACTION

    Check_AllowedToInit := Main.Check_PicAlphaConveyor_AllowedToInit;
    Check_AllowedToReceive := Main.Check_PicAlphaConveyor_AllowedToReceive;
    Check_AllowedToSend := Main.Check_PicAlphaConveyor_AllowedToSend;
    Check_FollowConveyor_InitCompleted := Main.Check_PicAlphaConveyor_FollowConveyor_InitCompleted;
    Check_PicAlpha_AutomaticExecuteCompleted := Main.Check_PicAlphaConveyor_PicAlpha_AutomaticExecuteCompleted;
    Check_FollowConveyor_AutomaticExecuteCompleted := Main.Check_PicAlphaConveyor_FollowConveyor_AutomaticExecuteCompleted;
    Check_EngineStop := MAIN.PPU_EngineStop;
    IF Check_EngineStop THEN
    	Motor.ACT_Stop();
    END_IF
END_FUNCTION_BLOCK

FUNCTION_BLOCK PositionTransmitter

    VAR_OUTPUT
        DI_PositionReached : BOOL;
    END_VAR

END_FUNCTION_BLOCK

FUNCTION_BLOCK Potentiometer

    VAR_OUTPUT
        AtStack : BOOL;
        AtConveyor : BOOL;
        AtStamp : BOOL;
    END_VAR

    VAR
        AI_Position : INT;
        delta : INT := 100;
        iPosStack : INT := 24310;
        iPosConveyor : INT := 15930;
        iPosStamp : INT := 7845;
    END_VAR

    IF((iPosStack-delta) < AI_Position AND AI_Position < (iPosStack+delta)) THEN
    	AtStack := TRUE;
    	AtConveyor := FALSE;
    	AtStamp := FALSE;
    ELSIF((iPosConveyor-delta) < AI_Position AND AI_Position < (iPosConveyor+delta)) THEN
    	AtStack := FALSE;
    	AtConveyor := TRUE;
    	AtStamp := FALSE;
    ELSIF((iPosStamp-delta) < AI_Position AND AI_Position < (iPosStamp+delta)) THEN
    	AtStack := FALSE;
    	AtConveyor := FALSE;
    	AtStamp := TRUE;
    ELSE
    	AtStack := FALSE;
    	AtConveyor := FALSE;
    	AtStamp := FALSE;
    END_IF
END_FUNCTION_BLOCK

FUNCTION_BLOCK PresenceSensor

    VAR
        DI_WPDetected : BOOL;
    END_VAR

END_FUNCTION_BLOCK

FUNCTION_BLOCK PressureSensor

    VAR
        AI_CurrentPressure : INT;
    END_VAR

END_FUNCTION_BLOCK

FUNCTION_BLOCK PressureSensor_4bar

    VAR
        DI_PressureReached : BOOL;
    END_VAR

END_FUNCTION_BLOCK

FUNCTION_BLOCK ProportionalValve

    VAR_INPUT
        AO_SetPressure : INT;
    END_VAR

END_FUNCTION_BLOCK

FUNCTION_BLOCK ProtectiveContact

    VAR
        DO_Plug : BOOL;
    END_VAR

END_FUNCTION_BLOCK

FUNCTION_BLOCK Ramp

    VAR_INPUT
        RampFull : PresenceSensor;
    END_VAR

END_FUNCTION_BLOCK

FUNCTION_BLOCK RefillConveyor

    VAR_INPUT
        PsBegining : PresenceSensor;
        PsSwitch : PresenceSensor;
        Switch : Switch;
        Motor : Motor;
        Check_AllowedToInit : BOOL;
        Check_AllowedToReceive : BOOL;
        Check_AllowedToSend : BOOL;
        Check_FollowConveyor_InitCompleted : BOOL;
        Check_FollowConveyor_AutomaticExecuteCompleted : BOOL;
        Check_EngineStop : BOOL;
        SFCReset : BOOL;
    END_VAR

    VAR_OUTPUT
        InitCompleted : BOOL;
        FollowConveyor_AllowedToInit : BOOL;
        FollowConveyor_AllowedToOperate : BOOL;
        AutomaticExecuteReceivingCompleted : BOOL;
        IsSending : BOOL;
        AutomaticExecuteSendingCompleted : BOOL;
        EmergencyHandled : BOOL;
    END_VAR

    VAR
        ConveyorSpeed : INT;
        NumberOfWPs : USINT;
        WPSeperated : BOOL;
        SFCInit : BOOL;
    END_VAR
    ACTION CountUp_WPNumber

        NumberOfWPs := NumberOfWPs+1;
    END_ACTION
    ACTION Reduce_WPNumber

        NumberOfWPs := NumberOfWPs-1;
    END_ACTION
    ACTION Reset_FollowConveyorAllowedToInit

        FollowConveyor_AllowedToInit := FALSE;
    END_ACTION
    ACTION Reset_FollowConveyorAllowedToOperate

        FollowConveyor_AllowedToOperate := FALSE;
    END_ACTION
    ACTION Reset_Variables

        InitCompleted := FALSE;
        FollowConveyor_AllowedToInit := FALSE;
        FollowConveyor_AllowedToOperate := FALSE;
        AutomaticExecuteReceivingCompleted := FALSE;
        AutomaticExecuteSendingCompleted := FALSE;
        NumberOfWPs := 0;
        WPSeperated := FALSE;
        Check_FollowConveyor_InitCompleted := FALSE;
        Check_AllowedToReceive := FALSE;
        Check_AllowedToSend := FALSE;
        Check_FollowConveyor_AutomaticExecuteCompleted := FALSE;
    END_ACTION
    ACTION Set_FollowConveyorAllowedToInit

        FollowConveyor_AllowedToInit := TRUE;
    END_ACTION
    ACTION Set_FollowConveyorAllowedToOperate

        FollowConveyor_AllowedToOperate := TRUE;
    END_ACTION
    ACTION ACT_SeperateWP

        INITIAL_STEP Init_ACT_SeperateWP : (*Local Id: 0 *)
        END_STEP

        STEP ExtendSwitch : (*Local Id: 3 *)
            Switch.ACT_Extend(N);
        END_STEP

        STEP RetractSwitch : (*Local Id: 6 *)
            Switch.ACT_Retract(N);
        END_STEP

        STEP WP_Seperated : (*Local Id: 9 *)
        END_STEP
        TRANSITION FROM (Init_ACT_SeperateWP) TO (ExtendSwitch) := (NOT WPSeperated AND NOT GVL.IsSFCResetting); END_TRANSITION
        TRANSITION FROM (ExtendSwitch) TO (RetractSwitch) := (Switch.Extended); END_TRANSITION
        TRANSITION FROM (RetractSwitch) TO (WP_Seperated) := (Switch.Retracted); END_TRANSITION
        TRANSITION FROM (WP_Seperated) TO (Init_ACT_SeperateWP) := (WPSeperated); END_TRANSITION
    END_ACTION
    ACTION ACT_AutomaticExecute

        INITIAL_STEP Init_ACT_AutomaticExecute : (*Local Id: 0 *)
        END_STEP

        STEP Choice_ReceivingSending : (*Local Id: 3 *)
        END_STEP

        STEP Interstep_Receiving : (*Local Id: 7 *)
        END_STEP

        STEP ConveyorForwards_Receiving : (*Local Id: 15 *)
            Motor.ACT_TurnClockwise(N);
        END_STEP

        STEP StopConveyor_Receiving : (*Local Id: 18 *)
        END_STEP

        STEP CountUpWPNumber : (*Local Id: 23 *)
            CountUp_WPNumber(N);
        END_STEP

        STEP ReceivingCompleted : (*Local Id: 26 *)
        END_STEP

        STEP Interstep_Sending : (*Local Id: 33 *)
        END_STEP

        STEP Set_IsSending : (*Local Id: 37 *)
        END_STEP

        STEP Check_ifStillAllowedToOperate : (*Local Id: 42 *)
        END_STEP

        STEP ConveyorForwards_Sending : (*Local Id: 49 *)
            Motor.ACT_TurnClockwise(N);
        END_STEP

        STEP SeperateWP : (*Local Id: 52 *)
            ACT_SeperateWP(N);
        END_STEP

        STEP StopConveyor_Sending : (*Local Id: 55 *)
        END_STEP

        STEP SortWP : (*Local Id: 61 *)
            Set_FollowConveyorAllowedToOperate(P0);
            Reset_FollowConveyorAllowedToOperate(P1);
        END_STEP

        STEP Receiving_again : (*Local Id: 62 *)
        END_STEP

        STEP ReduceWPNumber : (*Local Id: 69 *)
            Reduce_WPNumber(N);
        END_STEP

        STEP SendingCompleted : (*Local Id: 73 *)
        END_STEP
        TRANSITION FROM (StopConveyor_Sending) TO (SortWP, Receiving_again) := (Motor.Stopped); END_TRANSITION
        TRANSITION FROM (SortWP, Interstep_Receiving) TO (ReduceWPNumber) := (Check_FollowConveyor_AutomaticExecuteCompleted); END_TRANSITION
        TRANSITION FROM (Choice_ReceivingSending) TO (Interstep_Receiving) := (Check_AllowedToReceive); END_TRANSITION
        TRANSITION FROM (Choice_ReceivingSending) TO (Interstep_Sending) := (Check_AllowedToSend AND NumberOfWPs=3); END_TRANSITION
        TRANSITION FROM (Interstep_Receiving) TO (ConveyorForwards_Receiving) := (Check_AllowedToReceive AND Interstep_Receiving.t>T#100ms); END_TRANSITION
        TRANSITION FROM (Interstep_Receiving) TO (Init_ACT_AutomaticExecute) := (NOT Check_AllowedToReceive AND Interstep_Receiving.t>T#100ms); END_TRANSITION
        TRANSITION FROM (Interstep_Sending) TO (Set_IsSending) := (Check_AllowedToSend AND NumberOfWPs=3 AND Interstep_Sending.t>T#750ms); END_TRANSITION
        TRANSITION FROM (Interstep_Sending) TO (Init_ACT_AutomaticExecute) := ((NOT Check_AllowedToSend OR NOT NumberOfWPs=3) AND Interstep_Sending.t>T#750ms); END_TRANSITION
        TRANSITION FROM (ReduceWPNumber) TO (SendingCompleted) := (NumberOfWPs=0); END_TRANSITION
        TRANSITION FROM (ReduceWPNumber) TO (ConveyorForwards_Sending) := (NumberOfWPs>0); END_TRANSITION
        TRANSITION FROM (Interstep_Receiving) TO (ConveyorForwards_Receiving) := (Check_AllowedToReceive AND Interstep_Receiving.t>T#100ms); END_TRANSITION
        TRANSITION FROM (Check_ifStillAllowedToOperate) TO (ConveyorForwards_Sending) := (Check_AllowedToSend); END_TRANSITION
        TRANSITION FROM (SendingCompleted) TO (Init_ACT_AutomaticExecute) := (NOT IsSending AND AutomaticExecuteSendingCompleted); END_TRANSITION
        TRANSITION FROM (ReceivingCompleted) TO (Init_ACT_AutomaticExecute) := (AutomaticExecuteReceivingCompleted); END_TRANSITION
        TRANSITION FROM (SendingCompleted) TO (Init_ACT_AutomaticExecute) := (NOT IsSending AND AutomaticExecuteSendingCompleted); END_TRANSITION
        TRANSITION FROM (Init_ACT_AutomaticExecute) TO (Choice_ReceivingSending) := (NOT AutomaticExecuteReceivingCompleted AND NOT AutomaticExecuteSendingCompleted AND NOT GVL.IsSFCResetting); END_TRANSITION
        TRANSITION FROM (ConveyorForwards_Receiving) TO (StopConveyor_Receiving) := (Motor.TurningClockwise); END_TRANSITION
        TRANSITION FROM (StopConveyor_Receiving) TO (CountUpWPNumber) := (Motor.Stopped); END_TRANSITION
        TRANSITION FROM (CountUpWPNumber) TO (ReceivingCompleted) := (TRUE); END_TRANSITION
        TRANSITION FROM (Set_IsSending) TO (Check_ifStillAllowedToOperate) := (IsSending); END_TRANSITION
        TRANSITION FROM (ConveyorForwards_Sending) TO (SeperateWP) := (Motor.TurningClockwise); END_TRANSITION
        TRANSITION FROM (SeperateWP) TO (StopConveyor_Sending) := (WPSeperated); END_TRANSITION
        TRANSITION FROM (Receiving_again) TO (Interstep_Receiving) := (Check_AllowedToReceive); END_TRANSITION
    END_ACTION
    ACTION ACT_EmergencyStop

        INITIAL_STEP Init_ACT_EmergencyStop : (*Local Id: 0 *)
        END_STEP

        STEP ResetVariables : (*Local Id: 3 *)
            Reset_Variables(N);
        END_STEP

        STEP StopConveyor : (*Local Id: 6 *)
            Motor.ACT_Stop(N);
        END_STEP

        STEP RetractSwitch : (*Local Id: 9 *)
            Switch.ACT_Retract(N);
        END_STEP

        STEP RefillConveyor_EmergencyHandled : (*Local Id: 12 *)
        END_STEP
        TRANSITION FROM (Init_ACT_EmergencyStop) TO (ResetVariables) := (NOT EmergencyHandled AND NOT GVL.IsSFCResetting); END_TRANSITION
        TRANSITION FROM (ResetVariables) TO (StopConveyor) := (NOT InitCompleted AND NOT AutomaticExecuteReceivingCompleted); END_TRANSITION
        TRANSITION FROM (StopConveyor) TO (RetractSwitch) := (Motor.Stopped); END_TRANSITION
        TRANSITION FROM (RetractSwitch) TO (RefillConveyor_EmergencyHandled) := (Switch.Retracted); END_TRANSITION
        TRANSITION FROM (RefillConveyor_EmergencyHandled) TO (Init_ACT_EmergencyStop) := (EmergencyHandled); END_TRANSITION
    END_ACTION
    ACTION ACT_Init

        INITIAL_STEP Init_ACT_Init : (*Local Id: 0 *)
        END_STEP

        STEP Interstep : (*Local Id: 5 *)
        END_STEP

        STEP RetractSwitch : (*Local Id: 13 *)
            Switch.ACT_Retract(N);
        END_STEP

        STEP ConveyorForwards : (*Local Id: 16 *)
            Motor.ACT_TurnClockwise(N);
        END_STEP

        STEP StopConveyor : (*Local Id: 19 *)
        END_STEP

        STEP Init_Completed : (*Local Id: 24 *)
        END_STEP
        TRANSITION FROM (Interstep) TO (RetractSwitch) := (Check_AllowedToInit AND NOT InitCompleted AND Interstep.t>T#500ms); END_TRANSITION
        TRANSITION FROM (Interstep) TO (Init_ACT_Init) := ((NOT Check_AllowedToInit OR InitCompleted) AND Interstep.t>T#500ms); END_TRANSITION
        TRANSITION FROM (Interstep) TO (RetractSwitch) := (Check_AllowedToInit AND NOT InitCompleted AND Interstep.t>T#500ms); END_TRANSITION
        TRANSITION FROM (Init_ACT_Init) TO (Interstep) := (Check_AllowedToInit AND NOT InitCompleted AND NOT GVL.IsSFCResetting); END_TRANSITION
        TRANSITION FROM (RetractSwitch) TO (ConveyorForwards) := (Switch.Retracted); END_TRANSITION
        TRANSITION FROM (ConveyorForwards) TO (StopConveyor) := (Motor.TurningClockwise); END_TRANSITION
        TRANSITION FROM (StopConveyor) TO (Init_Completed) := (Motor.Stopped); END_TRANSITION
        TRANSITION FROM (Init_Completed) TO (Init_ACT_Init) := (InitCompleted); END_TRANSITION
    END_ACTION

    Check_AllowedToInit := Main.Check_RefillConveyor_AllowedToInit;
    Check_AllowedToReceive := Main.Check_RefillConveyor_AllowedToReceive;
    Check_AllowedToSend := Main.Check_RefillConveyor_AllowedToSend;
    Check_FollowConveyor_InitCompleted := Main.Check_RefillConveyor_FollowConveyor_InitCompleted;
    Check_FollowConveyor_AutomaticExecuteCompleted := Main.Check_RefillConveyor_FollowConveyor_AutomaticExecuteCompleted;
    Check_EngineStop := MAIN.PPU_EngineStop;
    IF Check_EngineStop THEN
    	Motor.ACT_Stop();
    END_IF
END_FUNCTION_BLOCK
